METHOD testIsEqualToIgnoreCase : BOOL
VAR_INPUT
	(* for the test it's the parameter ``stringToCheck`` *)
	{attribute 'TcEncoding' := 'UTF-8'}
	stringToTest 	:Tc2_System.T_MaxString;
	(* for the test it's the parameter ``expected`` *)
	{attribute 'TcEncoding' := 'UTF-8'}
	expectedString	:Tc2_System.T_MaxString;
END_VAR
VAR 
	(* just the expectation if the assertion to test must be worng or true *)
	assertionIsWrong				:BOOL;
	(* contains the format string for the test message *)
	message							:Tc2_System.T_MaxString;
	(* contains ´´stringToTest´´ in upper case *)
	upperStringToTest				:Tc2_System.T_MaxString;
	(* contains ´´expectedString´´ in upper case *)
	upperExpectedString				:Tc2_System.T_MaxString;
	(* used for placeholder string if stringToTest can't be printed *)
	stringToTestAsString 			:Tc2_System.T_MaxString;
	(* used for placeholder string if expectedString can't be printed *)
	expectedStringAsString 			:Tc2_System.T_MaxString;
	(* contains stringToTest in normalized form *)
	normalizedStringToTest			:Tc2_System.T_MaxString;
	(* contains expectedString in normalized form *)
	normalizedExpectedString		:Tc2_System.T_MaxString;
	(* contains stringToTest in normalized form in upper case*)
	normalizedUpperStringToTest		:Tc2_System.T_MaxString;
	(* contains expectedString in normalized form in upper case*)
	normalizedUpperExpectedString	:Tc2_System.T_MaxString;
	(* holds characterCount of ``stringToTest`` *)
	stringToTestCharacterCount		:UDINT;
	(* holds characterCount of ``expectedString`` *)
	expectedCharacterCount			:UDINT;
	(* TwinCAT printf with the test message *)
	messageStringBuilder			:Tc2_Utilities.FB_FormatString;
	(* hold stringToCheck before assertion *)
	stringToTestBeforeAssertion		:Tc2_System.T_MaxString;
	(* hold expectedString before assertion *)
	expectedStringBeforeAssertion	:Tc2_System.T_MaxString;
END_VAR
THIS^.assertorContainer.resetAssertor();

stringToTestBeforeAssertion := stringToTest;
expectedStringBeforeAssertion := expectedString;
stringToTestAsString := stringToTest;
expectedStringAsString := expectedString;
upperStringToTest := stringToTest;
upperExpectedString := expectedString;

// both Strings to upper case
CNM_UnicodeUtilities.UpperCaseUtf8(ADR(upperStringToTest));
CNM_UnicodeUtilities.UpperCaseUtf8(ADR(upperExpectedString));

CNM_UnicodeUtilities.GetUtf8StringLength(
	ADR(upperStringToTest),
	characterCount => stringToTestCharacterCount
);
CNM_UnicodeUtilities.GetUtf8StringLength(
	ADR(upperExpectedString),
	characterCount => expectedCharacterCount
);
assertionIsWrong := ((
		stringToTestCharacterCount <> expectedCharacterCount
	) OR (
		CNM_UnicodeUtilities.FindInUtf8String(
			ADR(upperStringToTest),
			ADR(upperExpectedString)
		) <> 1
	)
);

message := SEL(
	assertionIsWrong,
	'stringToCheck is $'%s$' expected is $'%s$' assertion must be TRUE', 
	'stringToCheck is $'%s$' expected is $'%s$' assertion must be FALSE'
);

IF (
		Tc2_Standard.LEN(stringToTest) = TO_UINT(Tc2_System.MAX_STRING_LENGTH)
) THEN
	stringToTestAsString := 'String with Tc2_System.MAX_STRING_LENGTH characters';
END_IF
IF (
		Tc2_Standard.LEN(expectedString) = TO_UINT(Tc2_System.MAX_STRING_LENGTH)
) THEN
	expectedStringAsString := 'String with Tc2_System.MAX_STRING_LENGTH characters';
END_IF

messageStringBuilder(
	sFormat := message,
	arg1 := THIS^.AnyToArg(stringToTestAsString),
	arg2 := THIS^.AnyToArg(expectedStringAsString)
);


THIS^.assertorContainer.assertor.assert.strings.unicode.isEqualTo(
	stringToCheck := stringToTest,
	expected := expectedString,
	ignoreCases := TRUE,
	normalizeStrings := FALSE,
	message			:= ''
);

THIS^.AssertEquals_BOOL(
	Expected 	:= assertionIsWrong,
	Actual 		:= THIS^.assertorContainer.wasAssertionWrong,
	Message 	:= messageStringBuilder.sOut
);

THIS^.AssertEquals_STRING(
	Expected 	:= stringToTestBeforeAssertion,
	Actual 		:= stringToTest,
	Message 	:= 'the assertion changed $'stringToTest$''
);

THIS^.AssertEquals_STRING(
	Expected 	:= expectedStringBeforeAssertion,
	Actual 		:= expectedString,
	Message 	:= 'the assertion changed $'expectedString$''
);

THIS^.assertorContainer.resetAssertor();

CNM_UnicodeUtilities.NormalizeUtf8String(
	utf8StringBuffer := ADR(stringToTest),
	bufferSize := Tc2_System.MAX_STRING_LENGTH + 1,
	normalizedStringBuffer := ADR(normalizedStringToTest),
	normalForm := CNM_UnicodeUtilities.NormalizationForm.NFD
);
CNM_UnicodeUtilities.NormalizeUtf8String(
	utf8StringBuffer := ADR(expectedString),
	bufferSize := Tc2_System.MAX_STRING_LENGTH + 1,
	normalizedStringBuffer := ADR(normalizedExpectedString),
	normalForm := CNM_UnicodeUtilities.NormalizationForm.NFD
);

normalizedUpperStringToTest := normalizedStringToTest;
normalizedUpperExpectedString := normalizedExpectedString;
CNM_UnicodeUtilities.UpperCaseUtf8(ADR(normalizedUpperStringToTest));
CNM_UnicodeUtilities.UpperCaseUtf8(ADR(normalizedUpperExpectedString));

CNM_UnicodeUtilities.GetUtf8StringLength(
	ADR(normalizedUpperStringToTest),
	characterCount => stringToTestCharacterCount
);
CNM_UnicodeUtilities.GetUtf8StringLength(
	ADR(normalizedUpperExpectedString),
	characterCount => expectedCharacterCount
);
assertionIsWrong := ((
		stringToTestCharacterCount <> expectedCharacterCount
	) OR (
		CNM_UnicodeUtilities.FindInUtf8String(
			ADR(normalizedUpperStringToTest),
			ADR(normalizedUpperExpectedString)
		) <> 1
	)
);

THIS^.assertorContainer.assertor.assert.strings.unicode.isEqualTo(
	stringToCheck := stringToTest,
	expected := expectedString,
	ignoreCases := TRUE,
	normalizeStrings := TRUE,
	message			:= ''
);

THIS^.AssertEquals_BOOL(
	Expected 	:= assertionIsWrong,
	Actual 		:= THIS^.assertorContainer.wasAssertionWrong,
	Message 	:= messageStringBuilder.sOut
);

THIS^.AssertEquals_STRING(
	Expected 	:= stringToTestBeforeAssertion,
	Actual 		:= stringToTest,
	Message 	:= 'the assertion changed $'stringToTest$''
);

THIS^.AssertEquals_STRING(
	Expected 	:= expectedStringBeforeAssertion,
	Actual 		:= expectedString,
	Message 	:= 'the assertion changed $'expectedString$''
);
END_METHOD

(*
short summary
==================
This test method tests ``assert.string.unicode.isNotEmpty``
method of CNM_AssertionInterfaces library with various inputs

.. <legal notes>

legal notes
=================
| SPDX-FileCopyrightText: © 2022 ekvip automation GmbH <info@ekvip.de>
| SPDX-License-Identifier: Apache-2.0
| For details check: Apache-2.0_

.. _Apache-2.0: https://www.apache.org/licenses/LICENSE-2.0

.. </legal notes>

*)


METHOD testIsNotEmpty : BOOL
VAR_INPUT
	(* for the test it's the parameter ``stringToCheck`` *)
	{attribute 'TcEncoding' := 'UTF-8'}
	stringToTest :Tc2_System.T_MaxString;
END_VAR
VAR 
	(* just the expectation if the assertion to test must be worng or true *)
	assertionIsWrong				:BOOL;
	(* contains the format string for the test message *)
	message							:Tc2_System.T_MaxString;
	(* used for placeholder string if stringToTest can't be printed *)
	stringToTestAsString 			:Tc2_System.T_MaxString;
	(* holds characterCount of ``stringToTest`` *)
	stringToTestCharacterCount		:UDINT;
	(* TwinCAT printf with the test message *)
	messageStringBuilder			:Tc2_Utilities.FB_FormatString;
	(* hold stringToCheck before assertion *)
	stringToTestBeforeAssertion		:Tc2_System.T_MaxString;
END_VAR
THIS^.assertorContainer.resetAssertor();

stringToTestBeforeAssertion := stringToTest;
stringToTestAsString := stringToTest;

CNM_UnicodeUtilities.GetUtf8StringLength(
	ADR(stringToTest),
	characterCount => stringToTestCharacterCount
);
assertionIsWrong :=  stringToTestCharacterCount = 0;

message := SEL(
	assertionIsWrong,
	'stringToCheck is $'%s$' assertion must be TRUE', 
	'stringToCheck is $'%s$' assertion must be FALSE'
);

IF (
		Tc2_Standard.LEN(stringToTest) = TO_UINT(Tc2_System.MAX_STRING_LENGTH)
) THEN
	stringToTestAsString := 'String with Tc2_System.MAX_STRING_LENGTH characters';
END_IF

messageStringBuilder(
	sFormat := message,
	arg1 := THIS^.AnyToArg(stringToTestAsString),
);


THIS^.assertorContainer.assertor.assert.strings.unicode.isNotEmpty(
	stringToCheck := stringToTest,
	message			:= ''
);

THIS^.AssertEquals_BOOL(
	Expected 	:= assertionIsWrong,
	Actual 		:= THIS^.assertorContainer.wasAssertionWrong,
	Message 	:= messageStringBuilder.sOut
);

THIS^.AssertEquals_STRING(
	Expected 	:= stringToTestBeforeAssertion,
	Actual 		:= stringToTest,
	Message 	:= 'the assertion changed $'stringToTest$''
);
END_METHOD

(*
short summary
==================
This test method tests ``assert.string.unicode.isNotEqualTo``
method of CNM_AssertionInterfaces library with various inputs

.. <legal notes>

legal notes
=================
| SPDX-FileCopyrightText: © 2022 ekvip automation GmbH <info@ekvip.de>
| SPDX-License-Identifier: Apache-2.0
| For details check: Apache-2.0_

.. _Apache-2.0: https://www.apache.org/licenses/LICENSE-2.0

.. </legal notes>

*)


METHOD testIsNotEqualTo : BOOL
VAR_INPUT
	(* for the test it's the parameter ``stringToCheck`` *)
	{attribute 'TcEncoding' := 'UTF-8'}
	stringToTest 	:Tc2_System.T_MaxString;
	(* for the test it's the parameter ``unexpected`` *)
	{attribute 'TcEncoding' := 'UTF-8'}
	expectedString :Tc2_System.T_MaxString;
END_VAR
VAR 
	(* just the expectation if the assertion to test must be worng or true *)
	assertionIsWrong				:BOOL;
	(* contains the format string for the test message *)
	message							:Tc2_System.T_MaxString;
	(* used for placeholder string if stringToTest can't be printed *)
	stringToTestAsString 			:Tc2_System.T_MaxString;
	(* used for placeholder string if expectedString can't be printed *)
	expectedStringAsString 			:Tc2_System.T_MaxString;
	(* contains stringToTest in normalized form *)
	normalizedStringToTest			:Tc2_System.T_MaxString;
	(* contains expectedString in normalized form *)
	normalizedExpectedString		:Tc2_System.T_MaxString;
	(* holds characterCount of ``stringToTest`` *)
	stringToTestCharacterCount		:UDINT;
	(* holds characterCount of ``expectedString`` *)
	expectedCharacterCount			:UDINT;
	(* TwinCAT printf with the test message *)
	messageStringBuilder			:Tc2_Utilities.FB_FormatString;
	(* hold stringToCheck before assertion *)
	stringToTestBeforeAssertion		:Tc2_System.T_MaxString;
	(* hold expectedString before assertion *)
	expectedStringBeforeAssertion	:Tc2_System.T_MaxString;
	expected: INT;
END_VAR
THIS^.assertorContainer.resetAssertor();

stringToTestBeforeAssertion := stringToTest;
expectedStringBeforeAssertion := expectedString;
stringToTestAsString := stringToTest;
expectedStringAsString := expectedString;

CNM_UnicodeUtilities.GetUtf8StringLength(
	ADR(stringToTest),
	characterCount => stringToTestCharacterCount
);
CNM_UnicodeUtilities.GetUtf8StringLength(
	ADR(expectedString),
	characterCount => expectedCharacterCount
);
assertionIsWrong := ((
		stringToTestCharacterCount = expectedCharacterCount
	) AND_THEN (
		CNM_UnicodeUtilities.FindInUtf8String(
			ADR(stringToTest),
			ADR(expectedString)
		) = 1
	)
);

message := SEL(
	assertionIsWrong,
	'stringToCheck is $'%s$' unexpected is $'%s$' assertion must be TRUE', 
	'stringToCheck is $'%s$' unexpected is $'%s$' assertion must be FALSE'
);

IF (
		Tc2_Standard.LEN(stringToTest) = TO_UINT(Tc2_System.MAX_STRING_LENGTH)
) THEN
	stringToTestAsString := 'String with Tc2_System.MAX_STRING_LENGTH characters';
END_IF
IF (
		Tc2_Standard.LEN(expectedString) = TO_UINT(Tc2_System.MAX_STRING_LENGTH)
) THEN
	expectedStringAsString := 'String with Tc2_System.MAX_STRING_LENGTH characters';
END_IF


messageStringBuilder(
	sFormat := message,
	arg1 := THIS^.AnyToArg(stringToTestAsString),
	arg2 := THIS^.AnyToArg(expectedStringAsString)
);


THIS^.assertorContainer.assertor.assert.strings.unicode.isNotEqualTo(
	stringToCheck := stringToTest,
	unexpected := expectedString,
	ignoreCases := FALSE,
	normalizeStrings := FALSE,
	message			:= ''
);

THIS^.AssertEquals_BOOL(
	Expected 	:= assertionIsWrong,
	Actual 		:= THIS^.assertorContainer.wasAssertionWrong,
	Message 	:= messageStringBuilder.sOut
);

THIS^.AssertEquals_STRING(
	Expected 	:= stringToTestBeforeAssertion,
	Actual 		:= stringToTest,
	Message 	:= 'the assertion changed $'stringToTest$''
);

THIS^.AssertEquals_STRING(
	Expected 	:= expectedStringBeforeAssertion,
	Actual 		:= expectedString,
	Message 	:= 'the assertion changed $'expectedString$''
);

THIS^.assertorContainer.resetAssertor();

CNM_UnicodeUtilities.NormalizeUtf8String(
	utf8StringBuffer := ADR(stringToTest),
	bufferSize := Tc2_System.MAX_STRING_LENGTH + 1,
	normalizedStringBuffer := ADR(normalizedStringToTest),
	normalForm := CNM_UnicodeUtilities.NormalizationForm.NFD
);
CNM_UnicodeUtilities.NormalizeUtf8String(
	utf8StringBuffer := ADR(expectedString),
	bufferSize := Tc2_System.MAX_STRING_LENGTH + 1,
	normalizedStringBuffer := ADR(normalizedExpectedString),
	normalForm := CNM_UnicodeUtilities.NormalizationForm.NFD
);

CNM_UnicodeUtilities.GetUtf8StringLength(
	ADR(normalizedStringToTest),
	characterCount => stringToTestCharacterCount
);
CNM_UnicodeUtilities.GetUtf8StringLength(
	ADR(normalizedExpectedString),
	characterCount => expectedCharacterCount
);
assertionIsWrong := ((
		stringToTestCharacterCount = expectedCharacterCount
	) AND (
		CNM_UnicodeUtilities.FindInUtf8String(
			ADR(normalizedStringToTest),
			ADR(normalizedExpectedString)
		) = 1
	)
);

THIS^.assertorContainer.assertor.assert.strings.unicode.isNotEqualTo(
	stringToCheck := stringToTest,
	unexpected := expectedString,
	ignoreCases := FALSE,
	normalizeStrings := TRUE,
	message			:= ''
);

THIS^.AssertEquals_BOOL(
	Expected 	:= assertionIsWrong,
	Actual 		:= THIS^.assertorContainer.wasAssertionWrong,
	Message 	:= messageStringBuilder.sOut
);

THIS^.AssertEquals_STRING(
	Expected 	:= stringToTestBeforeAssertion,
	Actual 		:= stringToTest,
	Message 	:= 'the assertion changed $'stringToTest$''
);

THIS^.AssertEquals_STRING(
	Expected 	:= expectedStringBeforeAssertion,
	Actual 		:= expectedString,
	Message 	:= 'the assertion changed $'expectedString$''
);
END_METHOD

(*
short summary
==================
This test method tests ``assert.string.unicode.isNotEqualTo``
method of CNM_AssertionInterfaces library with various inputs

.. <legal notes>

legal notes
=================
| SPDX-FileCopyrightText: © 2022 ekvip automation GmbH <info@ekvip.de>
| SPDX-License-Identifier: Apache-2.0
| For details check: Apache-2.0_

.. _Apache-2.0: https://www.apache.org/licenses/LICENSE-2.0

.. </legal notes>

*)


METHOD testIsNotEqualToIgnoreCase : BOOL
VAR_INPUT
	(* for the test it's the parameter ``stringToCheck`` *)
	{attribute 'TcEncoding' := 'UTF-8'}
	stringToTest 	:Tc2_System.T_MaxString;
	(* for the test it's the parameter ``unexpected`` *)
	{attribute 'TcEncoding' := 'UTF-8'}
	expectedString :Tc2_System.T_MaxString;
END_VAR
VAR 
	(* just the expectation if the assertion to test must be worng or true *)
	assertionIsWrong				:BOOL;
	(* contains the format string for the test message *)
	message							:Tc2_System.T_MaxString;
	(* contains ´´stringToTest´´ in upper case *)
	upperStringToTest				:Tc2_System.T_MaxString;
	(* contains ´´expectedString´´ in upper case *)
	upperExpectedString				:Tc2_System.T_MaxString;
	(* used for placeholder string if stringToTest can't be printed *)
	stringToTestAsString 			:Tc2_System.T_MaxString;
	(* used for placeholder string if expectedString can't be printed *)
	expectedStringAsString 			:Tc2_System.T_MaxString;
	(* contains stringToTest in normalized form *)
	normalizedStringToTest			:Tc2_System.T_MaxString;
	(* contains expectedString in normalized form *)
	normalizedExpectedString		:Tc2_System.T_MaxString;
	(* contains stringToTest in normalized form in upper case*)
	normalizedUpperStringToTest		:Tc2_System.T_MaxString;
	(* contains expectedString in normalized form in upper case*)
	normalizedUpperExpectedString	:Tc2_System.T_MaxString;
	(* holds characterCount of ``stringToTest`` *)
	stringToTestCharacterCount		:UDINT;
	(* holds characterCount of ``expectedString`` *)
	expectedCharacterCount			:UDINT;
	(* TwinCAT printf with the test message *)
	messageStringBuilder			:Tc2_Utilities.FB_FormatString;
	(* hold stringToCheck before assertion *)
	stringToTestBeforeAssertion		:Tc2_System.T_MaxString;
	(* hold expectedString before assertion *)
	expectedStringBeforeAssertion	:Tc2_System.T_MaxString;
END_VAR
THIS^.assertorContainer.resetAssertor();

stringToTestBeforeAssertion := stringToTest;
expectedStringBeforeAssertion := expectedString;
stringToTestAsString := stringToTest;
expectedStringAsString := expectedString;
upperStringToTest := stringToTest;
upperExpectedString := expectedString;

// both Strings to upper case
CNM_UnicodeUtilities.UpperCaseUtf8(ADR(upperStringToTest));
CNM_UnicodeUtilities.UpperCaseUtf8(ADR(upperExpectedString));

CNM_UnicodeUtilities.GetUtf8StringLength(
	ADR(upperStringToTest),
	characterCount => stringToTestCharacterCount
);
CNM_UnicodeUtilities.GetUtf8StringLength(
	ADR(upperExpectedString),
	characterCount => expectedCharacterCount
);
assertionIsWrong := ((
		stringToTestCharacterCount = expectedCharacterCount
	) AND (
		CNM_UnicodeUtilities.FindInUtf8String(
			ADR(upperStringToTest),
			ADR(upperExpectedString)
		) = 1
	)
);

message := SEL(
	assertionIsWrong,
	'stringToCheck is $'%s$' unexpected is $'%s$' assertion must be TRUE', 
	'stringToCheck is $'%s$' unexpected is $'%s$' assertion must be FALSE'
);

IF (
		Tc2_Standard.LEN(stringToTest) = TO_UINT(Tc2_System.MAX_STRING_LENGTH)
) THEN
	stringToTestAsString := 'String with Tc2_System.MAX_STRING_LENGTH characters';
END_IF
IF (
		Tc2_Standard.LEN(expectedString) = TO_UINT(Tc2_System.MAX_STRING_LENGTH)
) THEN
	expectedStringAsString := 'String with Tc2_System.MAX_STRING_LENGTH characters';
END_IF

messageStringBuilder(
	sFormat := message,
	arg1 := THIS^.AnyToArg(stringToTestAsString),
	arg2 := THIS^.AnyToArg(expectedStringAsString)
);


THIS^.assertorContainer.assertor.assert.strings.unicode.isNotEqualTo(
	stringToCheck := stringToTest,
	unexpected := expectedString,
	ignoreCases := TRUE,
	normalizeStrings := FALSE,
	message			:= ''
);

THIS^.AssertEquals_BOOL(
	Expected 	:= assertionIsWrong,
	Actual 		:= THIS^.assertorContainer.wasAssertionWrong,
	Message 	:= messageStringBuilder.sOut
);

THIS^.AssertEquals_STRING(
	Expected 	:= stringToTestBeforeAssertion,
	Actual 		:= stringToTest,
	Message 	:= 'the assertion changed $'stringToTest$''
);

THIS^.AssertEquals_STRING(
	Expected 	:= expectedStringBeforeAssertion,
	Actual 		:= expectedString,
	Message 	:= 'the assertion changed $'expectedString$''
);

THIS^.assertorContainer.resetAssertor();

CNM_UnicodeUtilities.NormalizeUtf8String(
	utf8StringBuffer := ADR(stringToTest),
	bufferSize := Tc2_System.MAX_STRING_LENGTH + 1,
	normalizedStringBuffer := ADR(normalizedStringToTest),
	normalForm := CNM_UnicodeUtilities.NormalizationForm.NFD
);
CNM_UnicodeUtilities.NormalizeUtf8String(
	utf8StringBuffer := ADR(expectedString),
	bufferSize := Tc2_System.MAX_STRING_LENGTH + 1,
	normalizedStringBuffer := ADR(normalizedExpectedString),
	normalForm := CNM_UnicodeUtilities.NormalizationForm.NFD
);

normalizedUpperStringToTest := normalizedStringToTest;
normalizedUpperExpectedString := normalizedExpectedString;
CNM_UnicodeUtilities.UpperCaseUtf8(ADR(normalizedUpperStringToTest));
CNM_UnicodeUtilities.UpperCaseUtf8(ADR(normalizedUpperExpectedString));

CNM_UnicodeUtilities.GetUtf8StringLength(
	ADR(normalizedUpperStringToTest),
	characterCount => stringToTestCharacterCount
);
CNM_UnicodeUtilities.GetUtf8StringLength(
	ADR(normalizedUpperExpectedString),
	characterCount => expectedCharacterCount
);
assertionIsWrong := ((
		stringToTestCharacterCount = expectedCharacterCount
	) AND (
		CNM_UnicodeUtilities.FindInUtf8String(
			ADR(normalizedUpperStringToTest),
			ADR(normalizedUpperExpectedString)
		) = 1
	)
);

THIS^.assertorContainer.assertor.assert.strings.unicode.isNotEqualTo(
	stringToCheck := stringToTest,
	unexpected := expectedString,
	ignoreCases := TRUE,
	normalizeStrings := TRUE,
	message			:= ''
);

THIS^.AssertEquals_BOOL(
	Expected 	:= assertionIsWrong,
	Actual 		:= THIS^.assertorContainer.wasAssertionWrong,
	Message 	:= messageStringBuilder.sOut
);

THIS^.AssertEquals_STRING(
	Expected 	:= stringToTestBeforeAssertion,
	Actual 		:= stringToTest,
	Message 	:= 'the assertion changed $'stringToTest$''
);

THIS^.AssertEquals_STRING(
	Expected 	:= expectedStringBeforeAssertion,
	Actual 		:= expectedString,
	Message 	:= 'the assertion changed $'expectedString$''
);
END_METHOD

(*
short summary
==================
This test method tests ``assert.string.unicode.lengthIsBetween``
method of CNM_AssertionInterfaces library with various inputs

.. <legal notes>

legal notes
=================
| SPDX-FileCopyrightText: © 2022 ekvip automation GmbH <info@ekvip.de>
| SPDX-License-Identifier: Apache-2.0
| For details check: Apache-2.0_

.. _Apache-2.0: https://www.apache.org/licenses/LICENSE-2.0

.. </legal notes>

*)


METHOD testLengthIsBetween : BOOL
VAR_INPUT
	(* for the test it's the parameter ``stringToCheck`` *)
	{attribute 'TcEncoding' := 'UTF-8'}
	stringToTest 			:Tc2_System.T_MaxString;
	(* for the test it's the parameter ``maxLength`` *)
	maxLength 				:UDINT;
	(* for the test it's the parameter ``minLength`` *)
	minLength 				:UDINT;
	(* UnicodeStringLengthUnit the input is tested for *)
	stringLengthUnit		:CNM_AssertionInterfaces.UnicodeStringLengthUnit;
	(* contains ``stringToTest`` in only ascii charachters for test output *)
	stringToTestPrintable 	:Tc2_System.T_MaxString := '';
END_VAR
VAR 
	(* just the expectation if the assertion to test must be worng or true *)
	assertionIsWrong				:BOOL;
	(* contains the format string for the test message *)
	message							:Tc2_System.T_MaxString;
	(* used for placeholder string if stringToTest can't be printed *)
	stringToTestAsString 			:Tc2_System.T_MaxString;
	(* holds string with current ´´stringLengthUnit´´ for the test message*)
	currentStringLengthUnit 		:Tc2_System.T_MaxString;
	(* TwinCAT printf with the test message *)
	messageStringBuilder			:Tc2_Utilities.FB_FormatString;
	(* length of current string to check in bytes *)
	stringToTestByteCount			:UDINT;
	(* length of current string to check in characters *)
	stringToTestCodePointCount		:UDINT;
	(* length of ´´stringToCheck´´ *)
	normalizedLength 				:UDINT;
	(* holds the normalized ´´stringToCheck´´ *)
	{attribute 'TcEncoding' := 'UTF-8'}
	normalizedStringToTest 			:Tc2_System.T_MaxString;
	(* width of ´´stringToCheck´´ *)
	stringToTestWidth 				:DINT;
	(* visible characters of ´´stringToCheck´´ *)
	stringToTestVisibleCharacters	:UDINT := 0;
	(* hold stringToCheck before assertion *)
	stringToTestBeforeAssertion		:Tc2_System.T_MaxString;
END_VAR
THIS^.assertorContainer.resetAssertor();

stringToTestBeforeAssertion := stringToTest;
stringToTestAsString := stringToTest;

CNM_UnicodeUtilities.GetUtf8StringLength(ADR(stringToTest), byteCount => stringToTestByteCount, characterCount => stringToTestCodePointCount,);
CNM_UnicodeUtilities.GetUtf8StringWidth(ADR(stringToTest), visibleCharacters => stringToTestVisibleCharacters, width => stringToTestWidth);

IF (
		Tc2_Standard.LEN(stringToTest) = TO_UINT(Tc2_System.MAX_STRING_LENGTH)
) THEN
	stringToTestAsString := 'String with Tc2_System.MAX_STRING_LENGTH characters';
END_IF
IF (
		LEN(stringToTestPrintable) <> 0
) THEN
	stringToTestAsString := stringToTestPrintable;
END_IF

CASE stringLengthUnit OF
	
CNM_AssertionInterfaces.UnicodeStringLengthUnit.BYTES:
	currentStringLengthUnit := 'BYTES';
	
	assertionIsWrong := ((stringToTestByteCount < minLength) OR ( stringToTestByteCount > maxLength ));
	
	message := SEL(
		assertionIsWrong,
		'stringToCheck is $'%s$' with maxLength %u and minLength %u assertion must be TRUE  (%S)', 
		'stringToCheck is $'%s$' with maxLength %u and minLength %u assertion must be FALSE  (%S)'
	);
	
	messageStringBuilder(
		sFormat := message,
		arg1 := THIS^.AnyToArg(stringToTestAsString),
		arg2 := THIS^.AnyToArg(maxLength),
		arg3 := THIS^.AnyToArg(minLength),
		arg4 := THIS^.AnyToArg(currentStringLengthUnit)
	);
	
	THIS^.assertorContainer.assertor.assert.strings.unicode.lengthIsBetween(
		stringToCheck := stringToTest,
		maxLength := maxLength,
		minLength := minLength,
		stringLengthUnit := CNM_AssertionInterfaces.UnicodeStringLengthUnit.BYTES,
		message			:= ''
	);
	
	THIS^.AssertEquals_BOOL(
		Expected 	:= assertionIsWrong,
		Actual 		:= THIS^.assertorContainer.wasAssertionWrong,
		Message 	:= messageStringBuilder.sOut
	);
	
	THIS^.AssertEquals_STRING(
		Expected 	:= stringToTestBeforeAssertion,
		Actual 		:= stringToTest,
		Message 	:= 'the assertion changed $'stringToTest$''
	);
	
CNM_AssertionInterfaces.UnicodeStringLengthUnit.CHARACTERS:	
	currentStringLengthUnit := 'CHARACTERS';
	THIS^.assertorContainer.resetAssertor();
	
	assertionIsWrong := ((
			stringToTestCodePointCount < minLength
		) OR (
			stringToTestCodePointCount > maxLength
		)
	);
	
	message := SEL(
		assertionIsWrong,
		'stringToCheck is $'%s$' with maxLength %u and minLength %u assertion must be TRUE  (%S)', 
		'stringToCheck is $'%s$' with maxLength %u and minLength %u assertion must be FALSE  (%S)'
	);
	
	   messageStringBuilder(
		sFormat := message,
		arg1 := THIS^.AnyToArg(stringToTestAsString),
		arg2 := THIS^.AnyToArg(maxLength),
		arg3 := THIS^.AnyToArg(minLength),
		arg4 := THIS^.AnyToArg(currentStringLengthUnit)
	);
	
	THIS^.assertorContainer.assertor.assert.strings.unicode.lengthIsBetween(
		stringToCheck := stringToTest,
		maxLength := maxLength,
		minLength := minLength,
		stringLengthUnit := CNM_AssertionInterfaces.UnicodeStringLengthUnit.CHARACTERS,
		message			:= ''
	);
	
	THIS^.AssertEquals_BOOL(
		Expected 	:= assertionIsWrong,
		Actual 		:= THIS^.assertorContainer.wasAssertionWrong,
		Message 	:= messageStringBuilder.sOut
	);
	
	THIS^.AssertEquals_STRING(
		Expected 	:= stringToTestBeforeAssertion,
		Actual 		:= stringToTest,
		Message 	:= 'the assertion changed $'stringToTest$''
	);
	
CNM_AssertionInterfaces.UnicodeStringLengthUnit.CHARACTERS_NFD:	
	currentStringLengthUnit := 'NFD';
	THIS^.assertorContainer.resetAssertor();
	
	CNM_UnicodeUtilities.NormalizeUtf8String(
		utf8StringBuffer := ADR(stringToTest),
		normalForm := CNM_UnicodeUtilities.NormalizationForm.NFD,
		normalizedStringBuffer := ADR(normalizedStringToTest),
		bufferSize := Tc2_System.MAX_STRING_LENGTH + 1,
		normalizedStringLength => normalizedLength
	);
	CNM_UnicodeUtilities.GetUtf8StringLength(
		stringAddress := ADR(normalizedStringToTest),
		characterCount => stringToTestCodePointCount
	);
		
	assertionIsWrong := ((
			stringToTestCodePointCount < minLength
		) OR (
			stringToTestCodePointCount > maxLength
		)
	);
	
	message := SEL(
		assertionIsWrong,
		'stringToCheck is $'%s$' with maxLength %u and minLength %u assertion must be TRUE  (%S)', 
		'stringToCheck is $'%s$' with maxLength %u and minLength %u assertion must be FALSE  (%S)'
	);
	
	messageStringBuilder(
		sFormat := message,
		arg1 := THIS^.AnyToArg(stringToTestAsString),
		arg2 := THIS^.AnyToArg(maxLength),
		arg3 := THIS^.AnyToArg(minLength),
		arg4 := THIS^.AnyToArg(currentStringLengthUnit)
	);
	
	THIS^.assertorContainer.assertor.assert.strings.unicode.lengthIsBetween(
		stringToCheck := stringToTest,
		maxLength := maxLength,
		minLength := minLength,
		stringLengthUnit := CNM_AssertionInterfaces.UnicodeStringLengthUnit.CHARACTERS_NFD,
		message			:= ''
	);
	
	THIS^.AssertEquals_BOOL(
		Expected 	:= assertionIsWrong,
		Actual 		:= THIS^.assertorContainer.wasAssertionWrong,
		Message 	:= messageStringBuilder.sOut
	);
	
	THIS^.AssertEquals_STRING(
		Expected 	:= stringToTestBeforeAssertion,
		Actual 		:= stringToTest,
		Message 	:= 'the assertion changed $'stringToTest$''
	);
	
CNM_AssertionInterfaces.UnicodeStringLengthUnit.CHARACTERS_NFC:	
	currentStringLengthUnit := 'NFC';
	THIS^.assertorContainer.resetAssertor();
	
	CNM_UnicodeUtilities.NormalizeUtf8String(
		utf8StringBuffer := ADR(stringToTest),
		normalForm := CNM_UnicodeUtilities.NormalizationForm.NFC,
		normalizedStringBuffer := ADR(normalizedStringToTest),
		bufferSize := Tc2_System.MAX_STRING_LENGTH + 1,
		normalizedStringLength => normalizedLength
	);
	CNM_UnicodeUtilities.GetUtf8StringLength(
		stringAddress := ADR(normalizedStringToTest),
		characterCount => stringToTestCodePointCount
	);
		
	assertionIsWrong := ((
			stringToTestCodePointCount < minLength
		) OR (
			stringToTestCodePointCount > maxLength
		)
	);
	
	message := SEL(
		assertionIsWrong,
		'stringToCheck is $'%s$' with maxLength %u and minLength %u assertion must be TRUE  (%S)', 
		'stringToCheck is $'%s$' with maxLength %u and minLength %u assertion must be FALSE  (%S)'
	);
	
	messageStringBuilder(
		sFormat := message,
		arg1 := THIS^.AnyToArg(stringToTestAsString),
		arg2 := THIS^.AnyToArg(maxLength),
		arg3 := THIS^.AnyToArg(minLength),
		arg4 := THIS^.AnyToArg(currentStringLengthUnit)
	);
	
	THIS^.assertorContainer.assertor.assert.strings.unicode.lengthIsBetween(
		stringToCheck := stringToTest,
		maxLength := maxLength,
		minLength := minLength,
		stringLengthUnit := CNM_AssertionInterfaces.UnicodeStringLengthUnit.CHARACTERS_NFC,
		message			:= ''
	);
	
	THIS^.AssertEquals_BOOL(
		Expected 	:= assertionIsWrong,
		Actual 		:= THIS^.assertorContainer.wasAssertionWrong,
		Message 	:= messageStringBuilder.sOut
	);
	
	THIS^.AssertEquals_STRING(
		Expected 	:= stringToTestBeforeAssertion,
		Actual 		:= stringToTest,
		Message 	:= 'the assertion changed $'stringToTest$''
	);
	
CNM_AssertionInterfaces.UnicodeStringLengthUnit.VISIBLE_CHARACTERS:	
	currentStringLengthUnit := 'VISIBLE_CHARACTERS';
	THIS^.assertorContainer.resetAssertor();
	
	assertionIsWrong := ((
			stringToTestVisibleCharacters < minLength
		) OR (
			stringToTestVisibleCharacters > maxLength
		)
	);
	
	message := SEL(
		assertionIsWrong,
		'stringToCheck is $'%s$' with maxLength %u and minLength %u assertion must be TRUE  (%S)', 
		'stringToCheck is $'%s$' with maxLength %u and minLength %u assertion must be FALSE  (%S)'
	);
	
	messageStringBuilder(
		sFormat := message,
		arg1 := THIS^.AnyToArg(stringToTestAsString),
		arg2 := THIS^.AnyToArg(maxLength),
		arg3 := THIS^.AnyToArg(minLength),
		arg4 := THIS^.AnyToArg(currentStringLengthUnit)
	);
	
	THIS^.assertorContainer.assertor.assert.strings.unicode.lengthIsBetween(
		stringToCheck := stringToTest,
		maxLength := maxLength,
		minLength := minLength,
		stringLengthUnit := CNM_AssertionInterfaces.UnicodeStringLengthUnit.VISIBLE_CHARACTERS,
		message			:= ''
	);
	
	THIS^.AssertEquals_BOOL(
		Expected 	:= assertionIsWrong,
		Actual 		:= THIS^.assertorContainer.wasAssertionWrong,
		Message 	:= messageStringBuilder.sOut
	);
	
	THIS^.AssertEquals_STRING(
		Expected 	:= stringToTestBeforeAssertion,
		Actual 		:= stringToTest,
		Message 	:= 'the assertion changed $'stringToTest$''
	);
	
CNM_AssertionInterfaces.UnicodeStringLengthUnit.WIDTH:	
	currentStringLengthUnit := 'WIDTH';
	THIS^.assertorContainer.resetAssertor();
	
	assertionIsWrong := ((
			TO_UDINT(stringToTestWidth) < minLength
		) OR (
			TO_UDINT(stringToTestWidth) > maxLength
		)
	);
	
	message := SEL(
		assertionIsWrong,
		'stringToCheck is $'%s$' with maxLength %u and minLength %u assertion must be TRUE  (%S)', 
		'stringToCheck is $'%s$' with maxLength %u and minLength %u assertion must be FALSE  (%S)'
	);
	
	messageStringBuilder(
		sFormat := message,
		arg1 := THIS^.AnyToArg(stringToTestAsString),
		arg2 := THIS^.AnyToArg(maxLength),
		arg3 := THIS^.AnyToArg(minLength),
		arg4 := THIS^.AnyToArg(currentStringLengthUnit)
	);
	
	THIS^.assertorContainer.assertor.assert.strings.unicode.lengthIsBetween(
		stringToCheck := stringToTest,
		maxLength := maxLength,
		minLength := minLength,
		stringLengthUnit := CNM_AssertionInterfaces.UnicodeStringLengthUnit.WIDTH,
		message			:= ''
	);
	
	THIS^.AssertEquals_BOOL(
		Expected 	:= assertionIsWrong,
		Actual 		:= THIS^.assertorContainer.wasAssertionWrong,
		Message 	:= messageStringBuilder.sOut
	);

	THIS^.AssertEquals_STRING(
		Expected 	:= stringToTestBeforeAssertion,
		Actual 		:= stringToTest,
		Message 	:= 'the assertion changed $'stringToTest$''
	);

END_CASE
END_METHOD

(*
short summary
==================
This test method tests ``assert.string.unicode.lengthIsExact``
method of CNM_AssertionInterfaces library with various inputs

.. <legal notes>

legal notes
=================
| SPDX-FileCopyrightText: © 2022 ekvip automation GmbH <info@ekvip.de>
| SPDX-License-Identifier: Apache-2.0
| For details check: Apache-2.0_

.. _Apache-2.0: https://www.apache.org/licenses/LICENSE-2.0

.. </legal notes>

*)


METHOD testLengthIsExact : BOOL
VAR_INPUT
	(* for the test it's the parameter ``stringToCheck`` *)
	{attribute 'TcEncoding' := 'UTF-8'}
	stringToTest 			:Tc2_System.T_MaxString;
	(* for the test it's the parameter ``expectedLength`` *)
	expectedLength			:UDINT;
	(* UnicodeStringLengthUnit the input is tested for *)
	stringLengthUnit		:CNM_AssertionInterfaces.UnicodeStringLengthUnit;
	(* contains ``stringToTest`` in only ascii charachters for test output *)
	stringToTestPrintable	:Tc2_System.T_MaxString := '';
END_VAR
VAR 
	(* just the expectation if the assertion to test must be worng or true *)
	assertionIsWrong				:BOOL;
	(* contains the format string for the test message *)
	message							:Tc2_System.T_MaxString;
	(* used for placeholder string if stringToTest can't be printed *)
	stringToTestAsString 			:Tc2_System.T_MaxString;
	(* holds string with current ´´stringLengthUnit´´ for the test message*)
	currentStringLengthUnit 		:Tc2_System.T_MaxString;
	(* TwinCAT printf with the test message *)
	messageStringBuilder			:Tc2_Utilities.FB_FormatString;
	(* length of current string to check in bytes *)
	stringToTestByteCount			:UDINT;
	(* length of current string to check in characters *)
	stringToTestCodePointCount		:UDINT;
	(* length of ´´stringToCheck´´ *)
	normalizedLength 				:UDINT;
	(* holds the normalized ´´stringToCheck´´ *)
	{attribute 'TcEncoding' := 'UTF-8'}
	normalizedStringToTest 			:Tc2_System.T_MaxString;
	(* width of ´´stringToCheck´´ *)
	stringToTestWidth 				:DINT;
	(* visible characters of ´´stringToCheck´´ *)
	stringToTestVisibleCharacters	:UDINT := 0;
	(* hold stringToCheck before assertion *)
	stringToTestBeforeAssertion		:Tc2_System.T_MaxString;
END_VAR
THIS^.assertorContainer.resetAssertor();

stringToTestBeforeAssertion := stringToTest;
stringToTestAsString := stringToTest;

CNM_UnicodeUtilities.GetUtf8StringLength(ADR(stringToTest), byteCount => stringToTestByteCount, characterCount => stringToTestCodePointCount,);
CNM_UnicodeUtilities.GetUtf8StringWidth(ADR(stringToTest), visibleCharacters => stringToTestVisibleCharacters, width => stringToTestWidth);

IF (
		Tc2_Standard.LEN(stringToTest) = TO_UINT(Tc2_System.MAX_STRING_LENGTH)
) THEN
	stringToTestAsString := 'String with Tc2_System.MAX_STRING_LENGTH characters';
END_IF
IF (
		LEN(stringToTestPrintable) <> 0
) THEN
	stringToTestAsString := stringToTestPrintable;
END_IF

CASE stringLengthUnit OF

CNM_AssertionInterfaces.UnicodeStringLengthUnit.BYTES:
	currentStringLengthUnit := 'BYTES';
	
	assertionIsWrong := stringToTestByteCount <> expectedLength;
	
	message := SEL(
		assertionIsWrong,
		'stringToCheck is $'%s$' with expectedLength %u assertion must be TRUE  (%S)', 
		'stringToCheck is $'%s$' with expectedLength %u assertion must be FALSE  (%S)'
	);
	
	messageStringBuilder(
		sFormat := message,
		arg1 := THIS^.AnyToArg(stringToTestAsString),
		arg2 := THIS^.AnyToArg(expectedLength),
		arg3 := THIS^.AnyToArg(currentStringLengthUnit)
	);
	
	THIS^.assertorContainer.assertor.assert.strings.unicode.lengthIsExact(
		stringToCheck := stringToTest,
		expectedLength := expectedLength,
		stringLengthUnit := CNM_AssertionInterfaces.UnicodeStringLengthUnit.BYTES,
		message			:= ''
	);
	
	THIS^.AssertEquals_BOOL(
		Expected 	:= assertionIsWrong,
		Actual 		:= THIS^.assertorContainer.wasAssertionWrong,
		Message 	:= messageStringBuilder.sOut
	);
	
	THIS^.AssertEquals_STRING(
		Expected 	:= stringToTestBeforeAssertion,
		Actual 		:= stringToTest,
		Message 	:= 'the assertion changed $'stringToTest$''
	);
	
CNM_AssertionInterfaces.UnicodeStringLengthUnit.CHARACTERS:	
	currentStringLengthUnit := 'CHARACTERS';
	
	assertionIsWrong := stringToTestCodePointCount <> expectedLength;
	
	message := SEL(
		assertionIsWrong,
		'stringToCheck is $'%s$' with expectedLength %u assertion must be TRUE  (%S)', 
		'stringToCheck is $'%s$' with expectedLength %u assertion must be FALSE  (%S)'
	);
	
	messageStringBuilder(
		sFormat := message,
		arg1 := THIS^.AnyToArg(stringToTestAsString),
		arg2 := THIS^.AnyToArg(expectedLength),
		arg3 := THIS^.AnyToArg(currentStringLengthUnit)
	);
	
	THIS^.assertorContainer.assertor.assert.strings.unicode.lengthIsExact(
		stringToCheck := stringToTest,
		expectedLength := expectedLength,
		stringLengthUnit := CNM_AssertionInterfaces.UnicodeStringLengthUnit.CHARACTERS,
		message			:= ''
	);
	
	THIS^.AssertEquals_BOOL(
		Expected 	:= assertionIsWrong,
		Actual 		:= THIS^.assertorContainer.wasAssertionWrong,
		Message 	:= messageStringBuilder.sOut
	);
	
	THIS^.AssertEquals_STRING(
		Expected 	:= stringToTestBeforeAssertion,
		Actual 		:= stringToTest,
		Message 	:= 'the assertion changed $'stringToTest$''
	);
	
CNM_AssertionInterfaces.UnicodeStringLengthUnit.CHARACTERS_NFD:	
	currentStringLengthUnit := 'NFD';
	
	CNM_UnicodeUtilities.NormalizeUtf8String(
		utf8StringBuffer := ADR(stringToTest),
		normalForm := CNM_UnicodeUtilities.NormalizationForm.NFD,
		normalizedStringBuffer := ADR(normalizedStringToTest),
		bufferSize := Tc2_System.MAX_STRING_LENGTH + 1,
		normalizedStringLength => normalizedLength
	);
	CNM_UnicodeUtilities.GetUtf8StringLength(
		stringAddress := ADR(normalizedStringToTest),
		characterCount => stringToTestCodePointCount
	);
		
	assertionIsWrong := stringToTestCodePointCount <> expectedLength;
	
	message := SEL(
		assertionIsWrong,
		'stringToCheck is $'%s$' with expectedLength %u assertion must be TRUE  (%S)', 
		'stringToCheck is $'%s$' with expectedLength %u assertion must be FALSE  (%S)'
	);
	
	messageStringBuilder(
		sFormat := message,
		arg1 := THIS^.AnyToArg(stringToTestAsString),
		arg2 := THIS^.AnyToArg(expectedLength),
		arg3 := THIS^.AnyToArg(currentStringLengthUnit)
	);
	
	THIS^.assertorContainer.assertor.assert.strings.unicode.lengthIsExact(
		stringToCheck := stringToTest,
		expectedLength := expectedLength,
		stringLengthUnit := CNM_AssertionInterfaces.UnicodeStringLengthUnit.CHARACTERS_NFD,
		message			:= ''
	);
	
	THIS^.AssertEquals_BOOL(
		Expected 	:= assertionIsWrong,
		Actual 		:= THIS^.assertorContainer.wasAssertionWrong,
		Message 	:= messageStringBuilder.sOut
	);
	
	THIS^.AssertEquals_STRING(
		Expected 	:= stringToTestBeforeAssertion,
		Actual 		:= stringToTest,
		Message 	:= 'the assertion changed $'stringToTest$''
	);
	
CNM_AssertionInterfaces.UnicodeStringLengthUnit.CHARACTERS_NFC:	
	currentStringLengthUnit := 'NFC';
	
	CNM_UnicodeUtilities.NormalizeUtf8String(
		utf8StringBuffer := ADR(stringToTest),
		normalForm := CNM_UnicodeUtilities.NormalizationForm.NFC,
		normalizedStringBuffer := ADR(normalizedStringToTest),
		bufferSize := Tc2_System.MAX_STRING_LENGTH + 1,
		normalizedStringLength => normalizedLength
	);
	CNM_UnicodeUtilities.GetUtf8StringLength(
		stringAddress := ADR(normalizedStringToTest),
		characterCount => stringToTestCodePointCount
	);
		
	assertionIsWrong := stringToTestCodePointCount <> expectedLength;
	
	message := SEL(
		assertionIsWrong,
		'stringToCheck is $'%s$' with expectedLength %u assertion must be TRUE  (%S)', 
		'stringToCheck is $'%s$' with expectedLength %u assertion must be FALSE  (%S)'
	);
	
	messageStringBuilder(
		sFormat := message,
		arg1 := THIS^.AnyToArg(stringToTestAsString),
		arg2 := THIS^.AnyToArg(expectedLength),
		arg3 := THIS^.AnyToArg(currentStringLengthUnit)
	);
	
	THIS^.assertorContainer.assertor.assert.strings.unicode.lengthIsExact(
		stringToCheck := stringToTest,
		expectedLength := expectedLength,
		stringLengthUnit := CNM_AssertionInterfaces.UnicodeStringLengthUnit.CHARACTERS_NFC,
		message			:= ''
	);
	
	THIS^.AssertEquals_BOOL(
		Expected 	:= assertionIsWrong,
		Actual 		:= THIS^.assertorContainer.wasAssertionWrong,
		Message 	:= messageStringBuilder.sOut
	);
	
	THIS^.AssertEquals_STRING(
		Expected 	:= stringToTestBeforeAssertion,
		Actual 		:= stringToTest,
		Message 	:= 'the assertion changed $'stringToTest$''
	);
	
CNM_AssertionInterfaces.UnicodeStringLengthUnit.VISIBLE_CHARACTERS:	
	currentStringLengthUnit := 'VISIBLE_CHARACTERS';
	
	assertionIsWrong := stringToTestVisibleCharacters <> expectedLength;
	
	message := SEL(
		assertionIsWrong,
		'stringToCheck is $'%s$' with expectedLength %u assertion must be TRUE  (%S)', 
		'stringToCheck is $'%s$' with expectedLength %u assertion must be FALSE  (%S)'
	);
	
	messageStringBuilder(
		sFormat := message,
		arg1 := THIS^.AnyToArg(stringToTestAsString),
		arg2 := THIS^.AnyToArg(expectedLength),
		arg3 := THIS^.AnyToArg(currentStringLengthUnit)
	);
	
	THIS^.assertorContainer.assertor.assert.strings.unicode.lengthIsExact(
		stringToCheck := stringToTest,
		expectedLength := expectedLength,
		stringLengthUnit := CNM_AssertionInterfaces.UnicodeStringLengthUnit.VISIBLE_CHARACTERS,
		message			:= ''
	);
	
	THIS^.AssertEquals_BOOL(
		Expected 	:= assertionIsWrong,
		Actual 		:= THIS^.assertorContainer.wasAssertionWrong,
		Message 	:= messageStringBuilder.sOut
	);
	
	THIS^.AssertEquals_STRING(
		Expected 	:= stringToTestBeforeAssertion,
		Actual 		:= stringToTest,
		Message 	:= 'the assertion changed $'stringToTest$''
	);
	
CNM_AssertionInterfaces.UnicodeStringLengthUnit.WIDTH:	
	currentStringLengthUnit := 'WIDTH';
	
	assertionIsWrong := TO_UDINT(stringToTestWidth) <> expectedLength;
	
	message := SEL(
		assertionIsWrong,
		'stringToCheck is $'%s$' with expectedLength %u assertion must be TRUE  (%S)', 
		'stringToCheck is $'%s$' with expectedLength %u assertion must be FALSE  (%S)'
	);
	
	messageStringBuilder(
		sFormat := message,
		arg1 := THIS^.AnyToArg(stringToTestAsString),
		arg2 := THIS^.AnyToArg(expectedLength),
		arg3 := THIS^.AnyToArg(currentStringLengthUnit)
	);
	
	THIS^.assertorContainer.assertor.assert.strings.unicode.lengthIsExact(
		stringToCheck := stringToTest,
		expectedLength := expectedLength,
		stringLengthUnit := CNM_AssertionInterfaces.UnicodeStringLengthUnit.WIDTH,
		message			:= ''
	);
	
	THIS^.AssertEquals_BOOL(
		Expected 	:= assertionIsWrong,
		Actual 		:= THIS^.assertorContainer.wasAssertionWrong,
		Message 	:= messageStringBuilder.sOut
	);

	THIS^.AssertEquals_STRING(
		Expected 	:= stringToTestBeforeAssertion,
		Actual 		:= stringToTest,
		Message 	:= 'the assertion changed $'stringToTest$''
	);

END_CASE
END_METHOD

(*
short summary
==================
This test method tests ``assert.string.unicode.lengthIsMax``
method of CNM_AssertionInterfaces library with various inputs

.. <legal notes>

legal notes
=================
| SPDX-FileCopyrightText: © 2022 ekvip automation GmbH <info@ekvip.de>
| SPDX-License-Identifier: Apache-2.0
| For details check: Apache-2.0_

.. _Apache-2.0: https://www.apache.org/licenses/LICENSE-2.0

.. </legal notes>

*)


METHOD testLengthIsMax : BOOL
VAR_INPUT
	(* for the test it's the parameter ``stringToCheck`` *)
	{attribute 'TcEncoding' := 'UTF-8'}
	stringToTest 			:Tc2_System.T_MaxString;
	(* for the test it's the parameter ``maxLength`` *)
	expectedLength			:UDINT;
	(* UnicodeStringLengthUnit the input is tested for *)
	stringLengthUnit		:CNM_AssertionInterfaces.UnicodeStringLengthUnit;
	(* contains ``stringToTest`` in only ascii charachters for test output *)
	stringToTestPrintable	:Tc2_System.T_MaxString := '';
END_VAR
VAR 
	(* just the expectation if the assertion to test must be worng or true *)
	assertionIsWrong				:BOOL;
	(* contains the format string for the test message *)
	message							:Tc2_System.T_MaxString;
	(* used for placeholder string if stringToTest can't be printed *)
	stringToTestAsString 			:Tc2_System.T_MaxString;
	(* holds string with current ´´stringLengthUnit´´ for the test message*)
	currentStringLengthUnit 		:Tc2_System.T_MaxString;
	(* TwinCAT printf with the test message *)
	messageStringBuilder			:Tc2_Utilities.FB_FormatString;
	(* length of current string to check in bytes *)
	stringToTestByteCount			:UDINT;
	(* length of current string to check in characters *)
	stringToTestCodePointCount		:UDINT;
	(* length of ´´stringToCheck´´ *)
	normalizedLength 				:UDINT;
	(* holds the normalized ´´stringToCheck´´ *)
	{attribute 'TcEncoding' := 'UTF-8'}
	normalizedStringToTest 			:Tc2_System.T_MaxString;
	(* width of ´´stringToCheck´´ *)
	stringToTestWidth 				:DINT;
	(* visible characters of ´´stringToCheck´´ *)
	stringToTestVisibleCharacters	:UDINT := 0;
	(* hold stringToCheck before assertion *)
	stringToTestBeforeAssertion		:Tc2_System.T_MaxString;
END_VAR
THIS^.assertorContainer.resetAssertor();

stringToTestBeforeAssertion := stringToTest;
stringToTestAsString := stringToTest;

CNM_UnicodeUtilities.GetUtf8StringLength(ADR(stringToTest), byteCount => stringToTestByteCount, characterCount => stringToTestCodePointCount,);
CNM_UnicodeUtilities.GetUtf8StringWidth(ADR(stringToTest), visibleCharacters => stringToTestVisibleCharacters, width => stringToTestWidth);

IF (
		Tc2_Standard.LEN(stringToTest) = TO_UINT(Tc2_System.MAX_STRING_LENGTH)
) THEN
	stringToTestAsString := 'String with Tc2_System.MAX_STRING_LENGTH characters';
END_IF
IF (
		LEN(stringToTestPrintable) <> 0
) THEN
	stringToTestAsString := stringToTestPrintable;
END_IF

CASE stringLengthUnit OF
	
CNM_AssertionInterfaces.UnicodeStringLengthUnit.BYTES:
	currentStringLengthUnit := 'BYTES';
	
	assertionIsWrong := stringToTestByteCount > expectedLength;
	
	message := SEL(
		assertionIsWrong,
		'stringToCheck is $'%s$' with expectedLength %u assertion must be TRUE  (%S)', 
		'stringToCheck is $'%s$' with expectedLength %u assertion must be FALSE  (%S)'
	);
	
	messageStringBuilder(
		sFormat := message,
		arg1 := THIS^.AnyToArg(stringToTestAsString),
		arg2 := THIS^.AnyToArg(expectedLength),
		arg3 := THIS^.AnyToArg(currentStringLengthUnit)
	);
	
	THIS^.assertorContainer.assertor.assert.strings.unicode.lengthIsMax(
		stringToCheck := stringToTest,
		maxLength := expectedLength,
		stringLengthUnit := CNM_AssertionInterfaces.UnicodeStringLengthUnit.BYTES,
		message			:= ''
	);
	
	THIS^.AssertEquals_BOOL(
		Expected 	:= assertionIsWrong,
		Actual 		:= THIS^.assertorContainer.wasAssertionWrong,
		Message 	:= messageStringBuilder.sOut
	);
	
	THIS^.AssertEquals_STRING(
		Expected 	:= stringToTestBeforeAssertion,
		Actual 		:= stringToTest,
		Message 	:= 'the assertion changed $'stringToTest$''
	);
	
CNM_AssertionInterfaces.UnicodeStringLengthUnit.CHARACTERS:	
	currentStringLengthUnit := 'CHARACTERS';
	THIS^.assertorContainer.resetAssertor();
	
	assertionIsWrong := stringToTestCodePointCount > expectedLength;
	
	message := SEL(
		assertionIsWrong,
		'stringToCheck is $'%s$' with expectedLength %u assertion must be TRUE  (%S)', 
		'stringToCheck is $'%s$' with expectedLength %u assertion must be FALSE  (%S)'
	);
	
	messageStringBuilder(
		sFormat := message,
		arg1 := THIS^.AnyToArg(stringToTestAsString),
		arg2 := THIS^.AnyToArg(expectedLength),
		arg3 := THIS^.AnyToArg(currentStringLengthUnit)
	);
	
	THIS^.assertorContainer.assertor.assert.strings.unicode.lengthIsMax(
		stringToCheck := stringToTest,
		maxLength := expectedLength,
		stringLengthUnit := CNM_AssertionInterfaces.UnicodeStringLengthUnit.CHARACTERS,
		message			:= ''
	);
	
	THIS^.AssertEquals_BOOL(
		Expected 	:= assertionIsWrong,
		Actual 		:= THIS^.assertorContainer.wasAssertionWrong,
		Message 	:= messageStringBuilder.sOut
	);
	
	THIS^.AssertEquals_STRING(
		Expected 	:= stringToTestBeforeAssertion,
		Actual 		:= stringToTest,
		Message 	:= 'the assertion changed $'stringToTest$''
	);
	
CNM_AssertionInterfaces.UnicodeStringLengthUnit.CHARACTERS_NFD:	
	currentStringLengthUnit := 'NFD';
	THIS^.assertorContainer.resetAssertor();
	
	CNM_UnicodeUtilities.NormalizeUtf8String(
		utf8StringBuffer := ADR(stringToTest),
		normalForm := CNM_UnicodeUtilities.NormalizationForm.NFD,
		normalizedStringBuffer := ADR(normalizedStringToTest),
		bufferSize := Tc2_System.MAX_STRING_LENGTH + 1,
		normalizedStringLength => normalizedLength
	);
	CNM_UnicodeUtilities.GetUtf8StringLength(
		stringAddress := ADR(normalizedStringToTest),
		characterCount => stringToTestCodePointCount
	);
		
	assertionIsWrong := stringToTestCodePointCount > expectedLength;
	
	message := SEL(
		assertionIsWrong,
		'stringToCheck is $'%s$' with expectedLength %u assertion must be TRUE  (%S)', 
		'stringToCheck is $'%s$' with expectedLength %u assertion must be FALSE  (%S)'
	);
	
	messageStringBuilder(
		sFormat := message,
		arg1 := THIS^.AnyToArg(stringToTestAsString),
		arg2 := THIS^.AnyToArg(expectedLength),
		arg3 := THIS^.AnyToArg(currentStringLengthUnit)
	);
	
	THIS^.assertorContainer.assertor.assert.strings.unicode.lengthIsMax(
		stringToCheck := stringToTest,
		maxLength := expectedLength,
		stringLengthUnit := CNM_AssertionInterfaces.UnicodeStringLengthUnit.CHARACTERS_NFD,
		message			:= ''
	);
	
	THIS^.AssertEquals_BOOL(
		Expected 	:= assertionIsWrong,
		Actual 		:= THIS^.assertorContainer.wasAssertionWrong,
		Message 	:= messageStringBuilder.sOut
	);
	
	THIS^.AssertEquals_STRING(
		Expected 	:= stringToTestBeforeAssertion,
		Actual 		:= stringToTest,
		Message 	:= 'the assertion changed $'stringToTest$''
	);
	
CNM_AssertionInterfaces.UnicodeStringLengthUnit.CHARACTERS_NFC:	
	currentStringLengthUnit := 'NFC';
	THIS^.assertorContainer.resetAssertor();
	
	CNM_UnicodeUtilities.NormalizeUtf8String(
		utf8StringBuffer := ADR(stringToTest),
		normalForm := CNM_UnicodeUtilities.NormalizationForm.NFC,
		normalizedStringBuffer := ADR(normalizedStringToTest),
		bufferSize := Tc2_System.MAX_STRING_LENGTH + 1,
		normalizedStringLength => normalizedLength
	);
	CNM_UnicodeUtilities.GetUtf8StringLength(
		stringAddress := ADR(normalizedStringToTest),
		characterCount => stringToTestCodePointCount
	);
		
	assertionIsWrong := stringToTestCodePointCount > expectedLength;
	
	message := SEL(
		assertionIsWrong,
		'stringToCheck is $'%s$' with expectedLength %u assertion must be TRUE  (%S)', 
		'stringToCheck is $'%s$' with expectedLength %u assertion must be FALSE  (%S)'
	);
	
	messageStringBuilder(
		sFormat := message,
		arg1 := THIS^.AnyToArg(stringToTestAsString),
		arg2 := THIS^.AnyToArg(expectedLength),
		arg3 := THIS^.AnyToArg(currentStringLengthUnit)
	);
	
	THIS^.assertorContainer.assertor.assert.strings.unicode.lengthIsMax(
		stringToCheck := stringToTest,
		maxLength := expectedLength,
		stringLengthUnit := CNM_AssertionInterfaces.UnicodeStringLengthUnit.CHARACTERS_NFC,
		message			:= ''
	);
	
	THIS^.AssertEquals_BOOL(
		Expected 	:= assertionIsWrong,
		Actual 		:= THIS^.assertorContainer.wasAssertionWrong,
		Message 	:= messageStringBuilder.sOut
	);
	
	THIS^.AssertEquals_STRING(
		Expected 	:= stringToTestBeforeAssertion,
		Actual 		:= stringToTest,
		Message 	:= 'the assertion changed $'stringToTest$''
	);
	
CNM_AssertionInterfaces.UnicodeStringLengthUnit.VISIBLE_CHARACTERS:	
	currentStringLengthUnit := 'VISIBLE_CHARACTERS';
	THIS^.assertorContainer.resetAssertor();
	
	assertionIsWrong := stringToTestVisibleCharacters > expectedLength;
	
	message := SEL(
		assertionIsWrong,
		'stringToCheck is $'%s$' with expectedLength %u assertion must be TRUE  (%S)', 
		'stringToCheck is $'%s$' with expectedLength %u assertion must be FALSE  (%S)'
	);
	
	messageStringBuilder(
		sFormat := message,
		arg1 := THIS^.AnyToArg(stringToTestAsString),
		arg2 := THIS^.AnyToArg(expectedLength),
		arg3 := THIS^.AnyToArg(currentStringLengthUnit)
	);
	
	THIS^.assertorContainer.assertor.assert.strings.unicode.lengthIsMax(
		stringToCheck := stringToTest,
		maxLength := expectedLength,
		stringLengthUnit := CNM_AssertionInterfaces.UnicodeStringLengthUnit.VISIBLE_CHARACTERS,
		message			:= ''
	);
	
	THIS^.AssertEquals_BOOL(
		Expected 	:= assertionIsWrong,
		Actual 		:= THIS^.assertorContainer.wasAssertionWrong,
		Message 	:= messageStringBuilder.sOut
	);
	
	THIS^.AssertEquals_STRING(
		Expected 	:= stringToTestBeforeAssertion,
		Actual 		:= stringToTest,
		Message 	:= 'the assertion changed $'stringToTest$''
	);
	
CNM_AssertionInterfaces.UnicodeStringLengthUnit.WIDTH:	
	currentStringLengthUnit := 'WIDTH';
	THIS^.assertorContainer.resetAssertor();
	
	assertionIsWrong := TO_UDINT(stringToTestWidth) > expectedLength;
	
	message := SEL(
		assertionIsWrong,
		'stringToCheck is $'%s$' with expectedLength %u assertion must be TRUE  (%S)', 
		'stringToCheck is $'%s$' with expectedLength %u assertion must be FALSE  (%S)'
	);
	
	messageStringBuilder(
		sFormat := message,
		arg1 := THIS^.AnyToArg(stringToTestAsString),
		arg2 := THIS^.AnyToArg(expectedLength),
		arg3 := THIS^.AnyToArg(currentStringLengthUnit)
	);
	
	THIS^.assertorContainer.assertor.assert.strings.unicode.lengthIsMax(
		stringToCheck := stringToTest,
		maxLength := expectedLength,
		stringLengthUnit := CNM_AssertionInterfaces.UnicodeStringLengthUnit.WIDTH,
		message			:= ''
	);
	
	THIS^.AssertEquals_BOOL(
		Expected 	:= assertionIsWrong,
		Actual 		:= THIS^.assertorContainer.wasAssertionWrong,
		Message 	:= messageStringBuilder.sOut
	);

	THIS^.AssertEquals_STRING(
		Expected 	:= stringToTestBeforeAssertion,
		Actual 		:= stringToTest,
		Message 	:= 'the assertion changed $'stringToTest$''
	);

END_CASE
END_METHOD

(*
short summary
==================
This test method tests ``assert.string.unicode.lengthIsMin``
method of CNM_AssertionInterfaces library with various inputs

.. <legal notes>

legal notes
=================
| SPDX-FileCopyrightText: © 2022 ekvip automation GmbH <info@ekvip.de>
| SPDX-License-Identifier: Apache-2.0
| For details check: Apache-2.0_

.. _Apache-2.0: https://www.apache.org/licenses/LICENSE-2.0

.. </legal notes>

*)


METHOD testLengthIsMin : BOOL
VAR_INPUT
	(* for the test it's the parameter ``stringToCheck`` *)
	{attribute 'TcEncoding' := 'UTF-8'}
	stringToTest 			:Tc2_System.T_MaxString;
	(* for the test it's the parameter ``minLength`` *)
	expectedLength 			:UDINT;
	(* UnicodeStringLengthUnit the input is tested for *)
	stringLengthUnit		:CNM_AssertionInterfaces.UnicodeStringLengthUnit;
	(* contains ``stringToTest`` in only ascii charachters for test output *)
	stringToTestPrintable	:Tc2_System.T_MaxString := '';
END_VAR
VAR 
	(* just the expectation if the assertion to test must be worng or true *)
	assertionIsWrong				:BOOL;
	(* contains the format string for the test message *)
	message							:Tc2_System.T_MaxString;
	(* used for placeholder string if stringToTest can't be printed *)
	stringToTestAsString 			:Tc2_System.T_MaxString;
	(* holds string with current ´´stringLengthUnit´´ for the test message*)
	currentStringLengthUnit 		:Tc2_System.T_MaxString;
	(* TwinCAT printf with the test message *)
	messageStringBuilder			:Tc2_Utilities.FB_FormatString;
	(* length of current string to check in bytes *)
	stringToTestByteCount			:UDINT;
	(* length of current string to check in characters *)
	stringToTestCodePointCount		:UDINT;
	(* length of ´´stringToCheck´´ *)
	normalizedLength 				:UDINT;
	(* holds the normalized ´´stringToCheck´´ *)
	{attribute 'TcEncoding' := 'UTF-8'}
	normalizedStringToTest 			:Tc2_System.T_MaxString;
	(* width of ´´stringToCheck´´ *)
	stringToTestWidth 				:DINT;
	(* visible characters of ´´stringToCheck´´ *)
	stringToTestVisibleCharacters	:UDINT := 0;
	(* hold stringToCheck before assertion *)
	stringToTestBeforeAssertion		:Tc2_System.T_MaxString;
END_VAR
THIS^.assertorContainer.resetAssertor();

stringToTestBeforeAssertion := stringToTest;
stringToTestAsString := stringToTest;

CNM_UnicodeUtilities.GetUtf8StringLength(ADR(stringToTest), byteCount => stringToTestByteCount, characterCount => stringToTestCodePointCount,);
CNM_UnicodeUtilities.GetUtf8StringWidth(ADR(stringToTest), visibleCharacters => stringToTestVisibleCharacters, width => stringToTestWidth);

IF (
		Tc2_Standard.LEN(stringToTest) = TO_UINT(Tc2_System.MAX_STRING_LENGTH)
) THEN
	stringToTestAsString := 'String with Tc2_System.MAX_STRING_LENGTH characters';
END_IF
IF (
		LEN(stringToTestPrintable) <> 0
) THEN
	stringToTestAsString := stringToTestPrintable;
END_IF

CASE stringLengthUnit OF
	
CNM_AssertionInterfaces.UnicodeStringLengthUnit.BYTES:
	currentStringLengthUnit := 'BYTES';
	
	assertionIsWrong := stringToTestByteCount < expectedLength;
	
	message := SEL(
		assertionIsWrong,
		'stringToCheck is $'%s$' with expectedLength %u assertion must be TRUE  (%S)', 
		'stringToCheck is $'%s$' with expectedLength %u assertion must be FALSE  (%S)'
	);
	
	messageStringBuilder(
		sFormat := message,
		arg1 := THIS^.AnyToArg(stringToTestAsString),
		arg2 := THIS^.AnyToArg(expectedLength),
		arg3 := THIS^.AnyToArg(currentStringLengthUnit)
	);
	
	THIS^.assertorContainer.assertor.assert.strings.unicode.lengthIsMin(
		stringToCheck := stringToTest,
		minLength := expectedLength,
		stringLengthUnit := CNM_AssertionInterfaces.UnicodeStringLengthUnit.BYTES,
		message			:= ''
	);
	
	THIS^.AssertEquals_BOOL(
		Expected 	:= assertionIsWrong,
		Actual 		:= THIS^.assertorContainer.wasAssertionWrong,
		Message 	:= messageStringBuilder.sOut
	);
	
	THIS^.AssertEquals_STRING(
		Expected 	:= stringToTestBeforeAssertion,
		Actual 		:= stringToTest,
		Message 	:= 'the assertion changed $'stringToTest$''
	);
	
CNM_AssertionInterfaces.UnicodeStringLengthUnit.CHARACTERS:	
	currentStringLengthUnit := 'CHARACTERS';
	THIS^.assertorContainer.resetAssertor();
	
	assertionIsWrong := stringToTestCodePointCount < expectedLength;
	
	message := SEL(
		assertionIsWrong,
		'stringToCheck is $'%s$' with expectedLength %u assertion must be TRUE  (%S)', 
		'stringToCheck is $'%s$' with expectedLength %u assertion must be FALSE  (%S)'
	);
	
	messageStringBuilder(
		sFormat := message,
		arg1 := THIS^.AnyToArg(stringToTestAsString),
		arg2 := THIS^.AnyToArg(expectedLength),
		arg3 := THIS^.AnyToArg(currentStringLengthUnit)
	);
	
	THIS^.assertorContainer.assertor.assert.strings.unicode.lengthIsMin(
		stringToCheck := stringToTest,
		minLength := expectedLength,
		stringLengthUnit := CNM_AssertionInterfaces.UnicodeStringLengthUnit.CHARACTERS,
		message			:= ''
	);
	
	THIS^.AssertEquals_BOOL(
		Expected 	:= assertionIsWrong,
		Actual 		:= THIS^.assertorContainer.wasAssertionWrong,
		Message 	:= messageStringBuilder.sOut
	);
	
	THIS^.AssertEquals_STRING(
		Expected 	:= stringToTestBeforeAssertion,
		Actual 		:= stringToTest,
		Message 	:= 'the assertion changed $'stringToTest$''
	);
	
CNM_AssertionInterfaces.UnicodeStringLengthUnit.CHARACTERS_NFD:	
	currentStringLengthUnit := 'NFD';
	THIS^.assertorContainer.resetAssertor();
	
	CNM_UnicodeUtilities.NormalizeUtf8String(
		utf8StringBuffer := ADR(stringToTest),
		normalForm := CNM_UnicodeUtilities.NormalizationForm.NFD,
		normalizedStringBuffer := ADR(normalizedStringToTest),
		bufferSize := Tc2_System.MAX_STRING_LENGTH + 1,
		normalizedStringLength => normalizedLength
	);
	CNM_UnicodeUtilities.GetUtf8StringLength(
		stringAddress := ADR(normalizedStringToTest),
		characterCount => stringToTestCodePointCount
	);
		
	assertionIsWrong := stringToTestCodePointCount < expectedLength;
	
	message := SEL(
		assertionIsWrong,
		'stringToCheck is $'%s$' with expectedLength %u assertion must be TRUE  (%S)', 
		'stringToCheck is $'%s$' with expectedLength %u assertion must be FALSE  (%S)'
	);
	
	messageStringBuilder(
		sFormat := message,
		arg1 := THIS^.AnyToArg(stringToTestAsString),
		arg2 := THIS^.AnyToArg(expectedLength),
		arg3 := THIS^.AnyToArg(currentStringLengthUnit)
	);
	
	THIS^.assertorContainer.assertor.assert.strings.unicode.lengthIsMin(
		stringToCheck := stringToTest,
		minLength := expectedLength,
		stringLengthUnit := CNM_AssertionInterfaces.UnicodeStringLengthUnit.CHARACTERS_NFD,
		message			:= ''
	);
	
	THIS^.AssertEquals_BOOL(
		Expected 	:= assertionIsWrong,
		Actual 		:= THIS^.assertorContainer.wasAssertionWrong,
		Message 	:= messageStringBuilder.sOut
	);
	
	THIS^.AssertEquals_STRING(
		Expected 	:= stringToTestBeforeAssertion,
		Actual 		:= stringToTest,
		Message 	:= 'the assertion changed $'stringToTest$''
	);
	
CNM_AssertionInterfaces.UnicodeStringLengthUnit.CHARACTERS_NFC:	
	currentStringLengthUnit := 'NFC';
	THIS^.assertorContainer.resetAssertor();
	
	CNM_UnicodeUtilities.NormalizeUtf8String(
		utf8StringBuffer := ADR(stringToTest),
		normalForm := CNM_UnicodeUtilities.NormalizationForm.NFC,
		normalizedStringBuffer := ADR(normalizedStringToTest),
		bufferSize := Tc2_System.MAX_STRING_LENGTH + 1,
		normalizedStringLength => normalizedLength
	);
	CNM_UnicodeUtilities.GetUtf8StringLength(
		stringAddress := ADR(normalizedStringToTest),
		characterCount => stringToTestCodePointCount
	);
		
	assertionIsWrong := stringToTestCodePointCount < expectedLength;
	
	message := SEL(
		assertionIsWrong,
		'stringToCheck is $'%s$' with expectedLength %u assertion must be TRUE  (%S)', 
		'stringToCheck is $'%s$' with expectedLength %u assertion must be FALSE  (%S)'
	);
	
	messageStringBuilder(
		sFormat := message,
		arg1 := THIS^.AnyToArg(stringToTestAsString),
		arg2 := THIS^.AnyToArg(expectedLength),
		arg3 := THIS^.AnyToArg(currentStringLengthUnit)
	);
	
	THIS^.assertorContainer.assertor.assert.strings.unicode.lengthIsMin(
		stringToCheck := stringToTest,
		minLength := expectedLength,
		stringLengthUnit := CNM_AssertionInterfaces.UnicodeStringLengthUnit.CHARACTERS_NFC,
		message			:= ''
	);
	
	THIS^.AssertEquals_BOOL(
		Expected 	:= assertionIsWrong,
		Actual 		:= THIS^.assertorContainer.wasAssertionWrong,
		Message 	:= messageStringBuilder.sOut
	);
	
	THIS^.AssertEquals_STRING(
		Expected 	:= stringToTestBeforeAssertion,
		Actual 		:= stringToTest,
		Message 	:= 'the assertion changed $'stringToTest$''
	);
	
CNM_AssertionInterfaces.UnicodeStringLengthUnit.VISIBLE_CHARACTERS:	
	currentStringLengthUnit := 'VISIBLE_CHARACTERS';
	THIS^.assertorContainer.resetAssertor();
	
	assertionIsWrong := stringToTestVisibleCharacters < expectedLength;
	
	message := SEL(
		assertionIsWrong,
		'stringToCheck is $'%s$' with expectedLength %u assertion must be TRUE  (%S)', 
		'stringToCheck is $'%s$' with expectedLength %u assertion must be FALSE  (%S)'
	);
	
	messageStringBuilder(
		sFormat := message,
		arg1 := THIS^.AnyToArg(stringToTestAsString),
		arg2 := THIS^.AnyToArg(expectedLength),
		arg3 := THIS^.AnyToArg(currentStringLengthUnit)
	);
	
	THIS^.assertorContainer.assertor.assert.strings.unicode.lengthIsMin(
		stringToCheck := stringToTest,
		minLength := expectedLength,
		stringLengthUnit := CNM_AssertionInterfaces.UnicodeStringLengthUnit.VISIBLE_CHARACTERS,
		message			:= ''
	);
	
	THIS^.AssertEquals_BOOL(
		Expected 	:= assertionIsWrong,
		Actual 		:= THIS^.assertorContainer.wasAssertionWrong,
		Message 	:= messageStringBuilder.sOut
	);
	
	THIS^.AssertEquals_STRING(
		Expected 	:= stringToTestBeforeAssertion,
		Actual 		:= stringToTest,
		Message 	:= 'the assertion changed $'stringToTest$''
	);
	
CNM_AssertionInterfaces.UnicodeStringLengthUnit.WIDTH:	
	currentStringLengthUnit := 'WIDTH';
	THIS^.assertorContainer.resetAssertor();
	
	assertionIsWrong := TO_UDINT(stringToTestWidth) < expectedLength;
	
	message := SEL(
		assertionIsWrong,
		'stringToCheck is $'%s$' with expectedLength %u assertion must be TRUE  (%S)', 
		'stringToCheck is $'%s$' with expectedLength %u assertion must be FALSE  (%S)'
	);
	
	messageStringBuilder(
		sFormat := message,
		arg1 := THIS^.AnyToArg(stringToTestAsString),
		arg2 := THIS^.AnyToArg(expectedLength),
		arg3 := THIS^.AnyToArg(currentStringLengthUnit)
	);
	
	THIS^.assertorContainer.assertor.assert.strings.unicode.lengthIsMin(
		stringToCheck := stringToTest,
		minLength := expectedLength,
		stringLengthUnit := CNM_AssertionInterfaces.UnicodeStringLengthUnit.WIDTH,
		message			:= ''
	);
	
	THIS^.AssertEquals_BOOL(
		Expected 	:= assertionIsWrong,
		Actual 		:= THIS^.assertorContainer.wasAssertionWrong,
		Message 	:= messageStringBuilder.sOut
	);
	
	THIS^.AssertEquals_STRING(
		Expected 	:= stringToTestBeforeAssertion,
		Actual 		:= stringToTest,
		Message 	:= 'the assertion changed $'stringToTest$''
	);
	
END_CASE
END_METHOD

(*
short summary
==================
This test method tests ``assert.string.unicode.startsWith``
method of CNM_AssertionInterfaces library with various inputs

.. <legal notes>

legal notes
=================
| SPDX-FileCopyrightText: © 2022 ekvip automation GmbH <info@ekvip.de>
| SPDX-License-Identifier: Apache-2.0
| For details check: Apache-2.0_

.. _Apache-2.0: https://www.apache.org/licenses/LICENSE-2.0

.. </legal notes>

*)


METHOD testStartsWith : BOOL
VAR_INPUT
	(* for the test it's the parameter ``stringToCheck`` *)
	{attribute 'TcEncoding' := 'UTF-8'}
	stringToTest 	:Tc2_System.T_MaxString;
	(* for the test it's the parameter ``end`` *)
	{attribute 'TcEncoding' := 'UTF-8'}
	expectedString 	:Tc2_System.T_MaxString;
END_VAR
VAR 
	(* just the expectation if the assertion to test must be worng or true *)
	assertionIsWrong				:BOOL;
	(* contains the format string for the test message *)
	message							:Tc2_System.T_MaxString;
	(* used for placeholder string if stringToTest can't be printed *)
	stringToTestAsString 			:Tc2_System.T_MaxString;
	(* used for placeholder string if expectedString can't be printed *)
	expectedStringAsString 			:Tc2_System.T_MaxString;
	(* contains stringToTest in normalized form *)
	normalizedStringToTest			:Tc2_System.T_MaxString;
	(* contains expectedString in normalized form *)
	normalizedExpectedString		:Tc2_System.T_MaxString;
	(* holds characterCount of ``expectedString`` *)
	expectedCharacterCount			:UDINT;
	(* TwinCAT printf with the test message *)
	messageStringBuilder			:Tc2_Utilities.FB_FormatString;
	(* hold stringToCheck before assertion *)
	stringToTestBeforeAssertion		:Tc2_System.T_MaxString;
	(* hold expectedString before assertion *)
	expectedStringBeforeAssertion	:Tc2_System.T_MaxString;
END_VAR
THIS^.assertorContainer.resetAssertor();

stringToTestBeforeAssertion := stringToTest;
expectedStringBeforeAssertion := expectedString;
stringToTestAsString := stringToTest;
expectedStringAsString := expectedString;

CNM_UnicodeUtilities.GetUtf8StringLength(
	ADR(expectedString),
	characterCount => expectedCharacterCount
);
assertionIsWrong := ((
		CNM_UnicodeUtilities.FindInUtf8String(
			ADR(stringToTest),
			ADR(expectedString),
		) <> 1
	) AND (
		expectedCharacterCount <> 0
	)
);

message := SEL(
	assertionIsWrong,
	'stringToCheck is $'%s$' start is $'%s$' assertion must be TRUE', 
	'stringToCheck is $'%s$' start is $'%s$' assertion must be FALSE'
);

IF (
		Tc2_Standard.LEN(stringToTest) = TO_UINT(Tc2_System.MAX_STRING_LENGTH)
) THEN
	stringToTestAsString := 'String with Tc2_System.MAX_STRING_LENGTH characters';
END_IF
IF (
		Tc2_Standard.LEN(expectedString) = TO_UINT(Tc2_System.MAX_STRING_LENGTH)
) THEN
	expectedStringAsString := 'String with Tc2_System.MAX_STRING_LENGTH characters';
END_IF

messageStringBuilder(
	sFormat := message,
	arg1 := THIS^.AnyToArg(stringToTestAsString),
	arg2 := THIS^.AnyToArg(expectedStringAsString)
);


THIS^.assertorContainer.assertor.assert.strings.unicode.startsWith(
	stringToCheck := stringToTest,
	start := expectedString,
	ignoreCases := FALSE,
	trim := FALSE,
	normalizeStrings := FALSE,
	message			:= ''
);

THIS^.AssertEquals_BOOL(
	Expected 	:= assertionIsWrong,
	Actual 		:= THIS^.assertorContainer.wasAssertionWrong,
	Message 	:= messageStringBuilder.sOut
);

THIS^.AssertEquals_STRING(
	Expected 	:= stringToTestBeforeAssertion,
	Actual 		:= stringToTest,
	Message 	:= 'the assertion changed $'stringToTest$''
);

THIS^.AssertEquals_STRING(
	Expected 	:= expectedStringBeforeAssertion,
	Actual 		:= expectedString,
	Message 	:= 'the assertion changed $'expectedString$''
);

THIS^.assertorContainer.resetAssertor();

CNM_UnicodeUtilities.NormalizeUtf8String(
	utf8StringBuffer := ADR(stringToTest),
	bufferSize := Tc2_System.MAX_STRING_LENGTH + 1,
	normalizedStringBuffer := ADR(normalizedStringToTest),
	normalForm := CNM_UnicodeUtilities.NormalizationForm.NFD
);
CNM_UnicodeUtilities.NormalizeUtf8String(
	utf8StringBuffer := ADR(expectedString),
	bufferSize := Tc2_System.MAX_STRING_LENGTH + 1,
	normalizedStringBuffer := ADR(normalizedExpectedString),
	normalForm := CNM_UnicodeUtilities.NormalizationForm.NFD
);

CNM_UnicodeUtilities.GetUtf8StringLength(
	ADR(normalizedExpectedString),
	characterCount => expectedCharacterCount
);
assertionIsWrong := ((
		CNM_UnicodeUtilities.FindInUtf8String(
			ADR(normalizedStringToTest),
			ADR(normalizedExpectedString),
		) <> 1
	) AND (
		expectedCharacterCount <> 0
	)
);

THIS^.assertorContainer.assertor.assert.strings.unicode.startsWith(
	stringToCheck := stringToTest,
	start := expectedString,
	ignoreCases := FALSE,
	trim		:= FALSE,
	normalizeStrings := TRUE,
	message			:= ''
);

THIS^.AssertEquals_BOOL(
	Expected 	:= assertionIsWrong,
	Actual 		:= THIS^.assertorContainer.wasAssertionWrong,
	Message 	:= messageStringBuilder.sOut
);

THIS^.AssertEquals_STRING(
	Expected 	:= stringToTestBeforeAssertion,
	Actual 		:= stringToTest,
	Message 	:= 'the assertion changed $'stringToTest$''
);

THIS^.AssertEquals_STRING(
	Expected 	:= expectedStringBeforeAssertion,
	Actual 		:= expectedString,
	Message 	:= 'the assertion changed $'expectedString$''
);
END_METHOD

(*
short summary
==================
This test method tests ``assert.string.unicode.startsWith``
method of CNM_AssertionInterfaces library with various inputs

.. <legal notes>

legal notes
=================
| SPDX-FileCopyrightText: © 2022 ekvip automation GmbH <info@ekvip.de>
| SPDX-License-Identifier: Apache-2.0
| For details check: Apache-2.0_

.. _Apache-2.0: https://www.apache.org/licenses/LICENSE-2.0

.. </legal notes>

*)


METHOD testStartsWithIgnoreCase : BOOL
VAR_INPUT
	(* for the test it's the parameter ``stringToCheck`` *)
	{attribute 'TcEncoding' := 'UTF-8'}
	stringToTest 	:Tc2_System.T_MaxString;
	(* for the test it's the parameter ``end`` *)
	{attribute 'TcEncoding' := 'UTF-8'}
	expectedString	:Tc2_System.T_MaxString;
END_VAR
VAR 
	(* just the expectation if the assertion to test must be worng or true *)
	assertionIsWrong				:BOOL;
	(* contains the format string for the test message *)
	message							:Tc2_System.T_MaxString;
	(* contains ´´stringToTest´´ in upper case *)
	upperStringToTest				:Tc2_System.T_MaxString;
	(* contains ´´expectedString´´ in upper case *)
	upperExpectedString				:Tc2_System.T_MaxString;
	(* used for placeholder string if stringToTest can't be printed *)
	stringToTestAsString 			:Tc2_System.T_MaxString;
	(* used for placeholder string if expectedString can't be printed *)
	expectedStringAsString 			:Tc2_System.T_MaxString;
	(* contains stringToTest in normalized form *)
	normalizedStringToTest			:Tc2_System.T_MaxString;
	(* contains expectedString in normalized form *)
	normalizedExpectedString		:Tc2_System.T_MaxString;
	(* contains stringToTest in normalized form in upper case*)
	normalizedUpperStringToTest		:Tc2_System.T_MaxString;
	(* contains expectedString in normalized form in upper case*)
	normalizedUpperExpectedString	:Tc2_System.T_MaxString;
	(* holds characterCount of ``expectedString`` *)
	expectedCharacterCount			:UDINT;
	(* TwinCAT printf with the test message *)
	messageStringBuilder			:Tc2_Utilities.FB_FormatString;
	(* hold stringToCheck before assertion *)
	stringToTestBeforeAssertion		:Tc2_System.T_MaxString;
	(* hold expectedString before assertion *)
	expectedStringBeforeAssertion	:Tc2_System.T_MaxString;
END_VAR
THIS^.assertorContainer.resetAssertor();

stringToTestBeforeAssertion := stringToTest;
expectedStringBeforeAssertion := expectedString;
stringToTestAsString := stringToTest;
expectedStringAsString := expectedString;
upperStringToTest := stringToTest;
upperExpectedString := expectedString;

// both Strings to upper case
CNM_UnicodeUtilities.UpperCaseUtf8(ADR(upperStringToTest));
CNM_UnicodeUtilities.UpperCaseUtf8(ADR(upperExpectedString));

CNM_UnicodeUtilities.GetUtf8StringLength(
	ADR(upperExpectedString),
	characterCount => expectedCharacterCount
);	
assertionIsWrong := ((
		CNM_UnicodeUtilities.FindInUtf8String(
			ADR(upperStringToTest),
			ADR(upperExpectedString)
		) <> 1 
	) AND (
		expectedCharacterCount <> 0
	)
);

message := SEL(
	assertionIsWrong,
	'stringToCheck is $'%s$' start is $'%s$' assertion must be TRUE', 
	'stringToCheck is $'%s$' start is $'%s$' assertion must be FALSE'
);

IF (
		Tc2_Standard.LEN(stringToTest) = TO_UINT(Tc2_System.MAX_STRING_LENGTH)
) THEN
	stringToTestAsString := 'String with Tc2_System.MAX_STRING_LENGTH characters';
END_IF
IF (
		Tc2_Standard.LEN(expectedString) = TO_UINT(Tc2_System.MAX_STRING_LENGTH)
) THEN
	expectedStringAsString := 'String with Tc2_System.MAX_STRING_LENGTH characters';
END_IF

messageStringBuilder(
	sFormat := message,
	arg1 := THIS^.AnyToArg(stringToTestAsString),
	arg2 := THIS^.AnyToArg(expectedStringAsString)
);


THIS^.assertorContainer.assertor.assert.strings.unicode.startsWith(
	stringToCheck := stringToTest,
	start := expectedString,
	ignoreCases := TRUE,
	trim := FALSE,
	message			:= ''
);

THIS^.AssertEquals_BOOL(
	Expected 	:= assertionIsWrong,
	Actual 		:= THIS^.assertorContainer.wasAssertionWrong,
	Message 	:= messageStringBuilder.sOut
);

THIS^.AssertEquals_STRING(
	Expected 	:= stringToTestBeforeAssertion,
	Actual 		:= stringToTest,
	Message 	:= 'the assertion changed $'stringToTest$''
);

THIS^.AssertEquals_STRING(
	Expected 	:= expectedStringBeforeAssertion,
	Actual 		:= expectedString,
	Message 	:= 'the assertion changed $'expectedString$''
);

THIS^.assertorContainer.resetAssertor();

CNM_UnicodeUtilities.NormalizeUtf8String(
	utf8StringBuffer := ADR(stringToTest),
	bufferSize := Tc2_System.MAX_STRING_LENGTH + 1,
	normalizedStringBuffer := ADR(normalizedStringToTest),
	normalForm := CNM_UnicodeUtilities.NormalizationForm.NFD
);
CNM_UnicodeUtilities.NormalizeUtf8String(
	utf8StringBuffer := ADR(expectedString),
	bufferSize := Tc2_System.MAX_STRING_LENGTH + 1,
	normalizedStringBuffer := ADR(normalizedExpectedString),
	normalForm := CNM_UnicodeUtilities.NormalizationForm.NFD
);

normalizedUpperStringToTest := normalizedStringToTest;
normalizedUpperExpectedString := normalizedExpectedString;
CNM_UnicodeUtilities.UpperCaseUtf8(ADR(normalizedUpperStringToTest));
CNM_UnicodeUtilities.UpperCaseUtf8(ADR(normalizedUpperExpectedString));


CNM_UnicodeUtilities.GetUtf8StringLength(
	ADR(normalizedUpperExpectedString),
	characterCount => expectedCharacterCount
);
assertionIsWrong := ((
		CNM_UnicodeUtilities.FindInUtf8String(
			ADR(normalizedUpperStringToTest),
			ADR(normalizedUpperExpectedString),
		) <> 1
	) AND (
		expectedCharacterCount <> 0
	)
);

THIS^.assertorContainer.assertor.assert.strings.unicode.startsWith(
	stringToCheck := stringToTest,
	start := expectedString,
	ignoreCases := TRUE,
	trim		:= FALSE,
	normalizeStrings := TRUE,
	message			:= ''
);

THIS^.AssertEquals_BOOL(
	Expected 	:= assertionIsWrong,
	Actual 		:= THIS^.assertorContainer.wasAssertionWrong,
	Message 	:= messageStringBuilder.sOut
);

THIS^.AssertEquals_STRING(
	Expected 	:= stringToTestBeforeAssertion,
	Actual 		:= stringToTest,
	Message 	:= 'the assertion changed $'stringToTest$''
);

THIS^.AssertEquals_STRING(
	Expected 	:= expectedStringBeforeAssertion,
	Actual 		:= expectedString,
	Message 	:= 'the assertion changed $'expectedString$''
);
END_METHOD

(*
short summary
==================
This test method tests ``assert.string.unicode.startsWith``
method of CNM_AssertionInterfaces library with various inputs

.. <legal notes>

legal notes
=================
| SPDX-FileCopyrightText: © 2022 ekvip automation GmbH <info@ekvip.de>
| SPDX-License-Identifier: Apache-2.0
| For details check: Apache-2.0_

.. _Apache-2.0: https://www.apache.org/licenses/LICENSE-2.0

.. </legal notes>

*)


METHOD testStartsWithTrim : BOOL
VAR_INPUT
	(* for the test it's the parameter ``stringToCheck`` *)
	{attribute 'TcEncoding' := 'UTF-8'}
	stringToTest 	:Tc2_System.T_MaxString;
	(* for the test it's the parameter ``end`` *)
	{attribute 'TcEncoding' := 'UTF-8'}
	expectedString 	:Tc2_System.T_MaxString;
END_VAR
VAR 
	(* just the expectation if the assertion to test must be worng or true *)
	assertionIsWrong				:BOOL;
	(* contains the format string for the test message *)
	message							:Tc2_System.T_MaxString;
	(* contains trimed ´´stringToTest´´ *)
	trimedStringToTest				:Tc2_System.T_MaxString;
	(* contains trimed ´´expectedString´´ *)
	trimedExpectedString			:Tc2_System.T_MaxString;
	(* used for placeholder string if stringToTest can't be printed *)
	stringToTestAsString 			:Tc2_System.T_MaxString;
	(* used for placeholder string if expectedString can't be printed *)
	expectedStringAsString 			:Tc2_System.T_MaxString;
	(* contains stringToTest in normalized form *)
	normalizedStringToTest			:Tc2_System.T_MaxString;
	(* contains expectedString in normalized form *)
	normalizedExpectedString		:Tc2_System.T_MaxString;
	(* contains stringToTest in normalized form trimed *)
	normalizedTrimedStringToTest	:Tc2_System.T_MaxString;
	(* contains expectedString in normalized form trimed *)
	normalizedTrimedExpectedString	:Tc2_System.T_MaxString;
	(* holds characterCount of ``expectedString`` *)
	expectedCharacterCount			:UDINT;
	(* TwinCAT printf with the test message *)
	messageStringBuilder			:Tc2_Utilities.FB_FormatString;
	(* hold stringToCheck before assertion *)
	stringToTestBeforeAssertion		:Tc2_System.T_MaxString;
	(* hold expectedString before assertion *)
	expectedStringBeforeAssertion	:Tc2_System.T_MaxString;
END_VAR
THIS^.assertorContainer.resetAssertor();

stringToTestBeforeAssertion := stringToTest;
expectedStringBeforeAssertion := expectedString;
stringToTestAsString := stringToTest;
expectedStringAsString := expectedString;
trimedStringToTest := stringToTest;
trimedExpectedString := expectedString;

// trim the left of both strings
CNM_UnicodeUtilities.TrimLeftUtf8String(ADR(trimedStringToTest));
CNM_UnicodeUtilities.TrimLeftUtf8String(ADR(trimedExpectedString));

CNM_UnicodeUtilities.GetUtf8StringLength(
	ADR(trimedExpectedString),
	characterCount => expectedCharacterCount
);
assertionIsWrong := ((
		CNM_UnicodeUtilities.FindInUtf8String(
			ADR(trimedStringToTest),
			ADR(trimedExpectedString),
		) <> 1
	) AND (
		expectedCharacterCount <> 0
	)
);

message := SEL(
	assertionIsWrong,
	'stringToCheck is $'%s$' start is $'%s$' assertion must be TRUE', 
	'stringToCheck is $'%s$' start is $'%s$' assertion must be FALSE'
);

IF (
		Tc2_Standard.LEN(stringToTest) = TO_UINT(Tc2_System.MAX_STRING_LENGTH)
) THEN
	stringToTestAsString := 'String with Tc2_System.MAX_STRING_LENGTH characters';
END_IF
IF (
		Tc2_Standard.LEN(expectedString) = TO_UINT(Tc2_System.MAX_STRING_LENGTH)
) THEN
	expectedStringAsString := 'String with Tc2_System.MAX_STRING_LENGTH characters';
END_IF

messageStringBuilder(
	sFormat := message,
	arg1 := THIS^.AnyToArg(stringToTestAsString),
	arg2 := THIS^.AnyToArg(expectedStringAsString)
);


THIS^.assertorContainer.assertor.assert.strings.unicode.startsWith(
	stringToCheck := stringToTest,
	start := expectedString,
	ignoreCases := FALSE,
	trim := TRUE,
	normalizeStrings := FALSE,
	message			:= ''
);

THIS^.AssertEquals_BOOL(
	Expected 	:= assertionIsWrong,
	Actual 		:= THIS^.assertorContainer.wasAssertionWrong,
	Message 	:= messageStringBuilder.sOut
);

THIS^.AssertEquals_STRING(
	Expected 	:= stringToTestBeforeAssertion,
	Actual 		:= stringToTest,
	Message 	:= 'the assertion changed $'stringToTest$''
);

THIS^.AssertEquals_STRING(
	Expected 	:= expectedStringBeforeAssertion,
	Actual 		:= expectedString,
	Message 	:= 'the assertion changed $'expectedString$''
);

THIS^.assertorContainer.resetAssertor();

CNM_UnicodeUtilities.NormalizeUtf8String(
	utf8StringBuffer := ADR(stringToTest),
	bufferSize := Tc2_System.MAX_STRING_LENGTH + 1,
	normalizedStringBuffer := ADR(normalizedStringToTest),
	normalForm := CNM_UnicodeUtilities.NormalizationForm.NFD
);
CNM_UnicodeUtilities.NormalizeUtf8String(
	utf8StringBuffer := ADR(expectedString),
	bufferSize := Tc2_System.MAX_STRING_LENGTH + 1,
	normalizedStringBuffer := ADR(normalizedExpectedString),
	normalForm := CNM_UnicodeUtilities.NormalizationForm.NFD
);

normalizedTrimedStringToTest := normalizedStringToTest;
normalizedTrimedExpectedString := normalizedExpectedString;
CNM_UnicodeUtilities.TrimLeftUtf8String(ADR(normalizedTrimedStringToTest));
CNM_UnicodeUtilities.TrimLeftUtf8String(ADR(normalizedTrimedExpectedString));

CNM_UnicodeUtilities.GetUtf8StringLength(
	ADR(normalizedTrimedExpectedString),
	characterCount => expectedCharacterCount
);
assertionIsWrong := ((
		CNM_UnicodeUtilities.FindInUtf8String(
			ADR(normalizedTrimedStringToTest),
			ADR(normalizedTrimedExpectedString),
		) <> 1
	) AND (
		expectedCharacterCount <> 0
	)
);

THIS^.assertorContainer.assertor.assert.strings.unicode.startsWith(
	stringToCheck := stringToTest,
	start := expectedString,
	ignoreCases := FALSE,
	trim		:= TRUE,
	normalizeStrings := TRUE,
	message			:= ''
);

THIS^.AssertEquals_BOOL(
	Expected 	:= assertionIsWrong,
	Actual 		:= THIS^.assertorContainer.wasAssertionWrong,
	Message 	:= messageStringBuilder.sOut
);

THIS^.AssertEquals_STRING(
	Expected 	:= stringToTestBeforeAssertion,
	Actual 		:= stringToTest,
	Message 	:= 'the assertion changed $'stringToTest$''
);

THIS^.AssertEquals_STRING(
	Expected 	:= expectedStringBeforeAssertion,
	Actual 		:= expectedString,
	Message 	:= 'the assertion changed $'expectedString$''
);
END_METHOD

END_FUNCTION_BLOCK

// ---- AssertionTester/AssertionTests/StringAssertions/classes/Windows125xStringAssertionTests.TcPOU

(*
short summary
==================
This class tests all methods of Windows125x string assertions
with various combinations of inputs and checks expected 
outputs are satisfied or not

.. <legal notes>

legal notes
=================
| SPDX-FileCopyrightText: © 2022 ekvip automation GmbH <info@ekvip.de>
| SPDX-License-Identifier: Apache-2.0
| For details check: Apache-2.0_

.. _Apache-2.0: https://www.apache.org/licenses/LICENSE-2.0

.. </legal notes>

methods and properties
======================

*)


FUNCTION_BLOCK Windows125xStringAssertionTests EXTENDS AbstractAssertorTest
VAR
	
END_VAR
VAR CONSTANT
	(* prefix to unify the test names *)
	TEST_NAME_PREFIX :STRING := 'assert.string.windows125x.';
	
END_VAR

THIS^.runIsEmpty();
THIS^.runIsNotEmpty();
THIS^.runContains();
THIS^.runContainsNo();
THIS^.runEndsWith();
THIS^.runStartsWith();
THIS^.runIsEqualTo();
THIS^.runIsNotEqualTo();
THIS^.runLengthIsBetween();
THIS^.runLengthIsExact();
THIS^.runLengthIsMax();
THIS^.runLengthIsMin();

(*

short summary
==================
This test method is a helper function to create a unified test name

.. <legal notes>

legal notes
=================
| SPDX-FileCopyrightText: © 2022 ekvip automation GmbH <info@ekvip.de>
| SPDX-License-Identifier: Apache-2.0
| For details check: Apache-2.0_

.. _Apache-2.0: https://www.apache.org/licenses/LICENSE-2.0

.. </legal notes>

parameters
==========

*)

METHOD PROTECTED getTestNameFor :Tc2_System.T_MaxString
VAR_INPUT
	(* name of the method to test, to create a unified test name *)
	nameOfMethodToTest	:Tc2_System.T_MaxString;
END_VAR
getTestNameFor := Tc2_Standard.CONCAT(THIS^.TEST_NAME_PREFIX, nameOfMethodToTest);
END_METHOD

(*
short summary
==================
This test method tests ``assert.string.windows125x.contains``
method of CNM_AssertionInterfaces library with various inputs

.. <legal notes>

legal notes
=================
| SPDX-FileCopyrightText: © 2022 ekvip automation GmbH <info@ekvip.de>
| SPDX-License-Identifier: Apache-2.0
| For details check: Apache-2.0_

.. _Apache-2.0: https://www.apache.org/licenses/LICENSE-2.0

.. </legal notes>

*)


METHOD runContains : BOOL
VAR_INPUT
END_VAR
RETURN (NOT TcUnit.TEST_ORDERED(THIS^.getTestNameFor('contains')));

THIS^.testContains(
	stringToTest := '',
	expectedString := ''
);
THIS^.testContains(
	stringToTest := 'not empty',
	expectedString := ''
);
THIS^.testContains(
	stringToTest := '',
	expectedString := 'not empty'
);
THIS^.testContains(
	stringToTest := 'not empty',
	expectedString := 'not empty'
);
THIS^.testContains(
	stringToTest := '{|}~',
	expectedString := '3649213469328'
);
THIS^.testContains(
	stringToTest := '1one!',
	expectedString := '1'
);
THIS^.testContains(
	stringToTest := '1one!',
	expectedString := 'one'
);
THIS^.testContains(
	stringToTest := '1one!',
	expectedString := '!'
);
THIS^.testContains(
	stringToTest := '$40$n$t$$$"$'',
	expectedString := '$n$t'
);
THIS^.testContains(
	stringToTest := '$80$8C$A9$B9$C6$D4$F4$7E',
	expectedString := '$B9$C6$D4'
);
THIS^.testContains(
	stringToTest := '$80$8C$A9$B9$C6$D4$F4$7E',
	expectedString := '$80$B9$C6$D4'
);
THIS^.testContains(
	stringToTest := 'frontmiddleback',
	expectedString := 'back'
);
THIS^.testContains(
	stringToTest := 'frontmiddleback',
	expectedString := 'frontmiddlebackfront'
);
THIS^.testContains(
	stringToTest := 'backfrontmiddle',
	expectedString := 'backmiddle'
);
THIS^.testContains(
	stringToTest := 'J;%_iTxQSk?6GfWewt}yMKh1)VXqPA@P1YQ:{EAg:8VJ,/FM;j)xJ[[AvYp/}}SzEgtfYS,1K0.5VtA+VJrB(p#55h2z##mw#F)Y@P6Jz9G@6vb=x#E!cYk(Svr@S*KiPJr1VZ6AjrNback4G=vBJd.E:=,k3!wmuGDe#ZKMD#Vx%?M_0&L0#vT]J,+)ZvU{w%8X0=:XzthmT0VG0QrwpXXCWpFxu6[b!c.BunYYfLQi.,?ut?-{jrC1phTHL)y',
	expectedString := 'J;%_iTxQSk?6GfWewt}yMKh1)VXqPA@P1YQ:{EAg:8VJ,/FM;j)xJ[[AvYp/}}SzEgtfYS,1K0.5VtA+VJrB(p#55h2z##mw#F)Y@P6Jz9G@6vb=x#E!cYk(Svr@S*KiPJr1VZ6AjrNback4G=vBJd.E:=,k3!wmuGDe#ZKMD#Vx%?M_0&L0#vT]J,+)ZvU{w%8X0=:XzthmT0VG0QrwpXXCWpFxu6[b!c.BunYYfLQi.,?ut?-{jrC1phTHL)y'
);
THIS^.testContains(
	stringToTest := 'J;%_iTxQSk?6GfWewt}yMKh1)VXqPA@P1YQ:{EAg:8VJ,/FM;j)xJ[[AvYp/}}SzEgtfYS,1K0.5VtA+VJrB(p#55h2z##mw#F)Y@P6Jz9G@6vb=x#E!cYk(Svr@S*KiPJr1VZ6AjrNback4G=vBJd.E:=,k3!wmuGDe#ZKMD#Vx%?M_0&L0#vT]J,+)ZvU{w%8X0=:XzthmT0VG0QrwpXXCWpFxu6[b!c.BunYYfLQi.,?ut?-{jrC1phTHL)y',
	expectedString := 'J;%_iTxQSk?6GfWewt}yMKh1)VXqPA@P1YQ:{EAg:8VJ,/FM;j)xJ[[AvYp/}}SzEgtfYS,1K0.5VtA+VJrB(p#55h2z##mw#F)Y@P6Jz9G@6vb=x#E!cYk(Svr@S*KiPJr1VZ6AjrNback4G=vBJd.E:=,k3!wmuGDe#ZKMD#Vx%?M_0&L0#vT]J,+)ZvU{w%8X0=:XzthmT0VG0QrwpXXCWpFxu6[b!c.BunYYfLQi.,?ut?-{jrC1phTHL)x'
);

THIS^.testContainsIgnoreCase(
	stringToTest := 'UPPERCASE',
	expectedString := 'CASE'
);
THIS^.testContainsIgnoreCase(
	stringToTest := 'lowercase',
	expectedString := 'case'
);
THIS^.testContainsIgnoreCase(
	stringToTest := 'UPPERCASE',
	expectedString := 'case'
);
THIS^.testContainsIgnoreCase(
	stringToTest := 'lowercase',
	expectedString := 'CASE'
);
THIS^.testContainsIgnoreCase(
	stringToTest := 'lower',
	expectedString := 'UPPER'
);
THIS^.testContainsIgnoreCase(
	stringToTest := 'lowercase$80$B9$C6$D4',
	expectedString := 'CASE$80$B9$C6$D4'
);

TcUnit.TEST_FINISHED();
END_METHOD

(*
short summary
==================
This test method tests ``assert.string.windows125x.containsNo``
method of CNM_AssertionInterfaces library with various inputs

.. <legal notes>

legal notes
=================
| SPDX-FileCopyrightText: © 2022 ekvip automation GmbH <info@ekvip.de>
| SPDX-License-Identifier: Apache-2.0
| For details check: Apache-2.0_

.. _Apache-2.0: https://www.apache.org/licenses/LICENSE-2.0

.. </legal notes>

*)


METHOD runContainsNo : BOOL
RETURN (NOT TcUnit.TEST_ORDERED(THIS^.getTestNameFor('containsNo')));

THIS^.testContainsNo(
	stringToTest := '',
	expectedString := ''
);
THIS^.testContainsNo(
	stringToTest := 'not empty',
	expectedString := ''
);
THIS^.testContainsNo(
	stringToTest := '',
	expectedString := 'not empty'
);
THIS^.testContainsNo(
	stringToTest := 'not empty',
	expectedString := 'not empty'
);
THIS^.testContainsNo(
	stringToTest := '{|}~',
	expectedString := '3649213469328'
);
THIS^.testContainsNo(
	stringToTest := '1one!',
	expectedString := '1'
);
THIS^.testContainsNo(
	stringToTest := '1one!',
	expectedString := 'one'
);
THIS^.testContainsNo(
	stringToTest := '1one!',
	expectedString := '!'
);
THIS^.testContainsNo(
	stringToTest := '$40$n$t$$$"$'',
	expectedString := '$n$t'
);
THIS^.testContainsNo(
	stringToTest := '$80$8C$A9$B9$C6$D4$F4$7E',
	expectedString := '$B9$C6$D4'
);
THIS^.testContainsNo(
	stringToTest := '$80$8C$A9$B9$C6$D4$F4$7E',
	expectedString := '$80$B9$C6$D4'
);
THIS^.testContainsNo(
	stringToTest := 'frontmiddleback',
	expectedString := 'back'
);
THIS^.testContainsNo(
	stringToTest := 'frontmiddleback',
	expectedString := 'frontmiddlebackfront'
);
THIS^.testContainsNo(
	stringToTest := 'backfrontmiddle',
	expectedString := 'backmiddle'
);
THIS^.testContainsNo(
	stringToTest := 'J;%_iTxQSk?6GfWewt}yMKh1)VXqPA@P1YQ:{EAg:8VJ,/FM;j)xJ[[AvYp/}}SzEgtfYS,1K0.5VtA+VJrB(p#55h2z##mw#F)Y@P6Jz9G@6vb=x#E!cYk(Svr@S*KiPJr1VZ6AjrNback4G=vBJd.E:=,k3!wmuGDe#ZKMD#Vx%?M_0&L0#vT]J,+)ZvU{w%8X0=:XzthmT0VG0QrwpXXCWpFxu6[b!c.BunYYfLQi.,?ut?-{jrC1phTHL)y',
	expectedString := 'J;%_iTxQSk?6GfWewt}yMKh1)VXqPA@P1YQ:{EAg:8VJ,/FM;j)xJ[[AvYp/}}SzEgtfYS,1K0.5VtA+VJrB(p#55h2z##mw#F)Y@P6Jz9G@6vb=x#E!cYk(Svr@S*KiPJr1VZ6AjrNback4G=vBJd.E:=,k3!wmuGDe#ZKMD#Vx%?M_0&L0#vT]J,+)ZvU{w%8X0=:XzthmT0VG0QrwpXXCWpFxu6[b!c.BunYYfLQi.,?ut?-{jrC1phTHL)y'
);
THIS^.testContainsNo(
	stringToTest := 'J;%_iTxQSk?6GfWewt}yMKh1)VXqPA@P1YQ:{EAg:8VJ,/FM;j)xJ[[AvYp/}}SzEgtfYS,1K0.5VtA+VJrB(p#55h2z##mw#F)Y@P6Jz9G@6vb=x#E!cYk(Svr@S*KiPJr1VZ6AjrNback4G=vBJd.E:=,k3!wmuGDe#ZKMD#Vx%?M_0&L0#vT]J,+)ZvU{w%8X0=:XzthmT0VG0QrwpXXCWpFxu6[b!c.BunYYfLQi.,?ut?-{jrC1phTHL)y',
	expectedString := 'J;%_iTxQSk?6GfWewt}yMKh1)VXqPA@P1YQ:{EAg:8VJ,/FM;j)xJ[[AvYp/}}SzEgtfYS,1K0.5VtA+VJrB(p#55h2z##mw#F)Y@P6Jz9G@6vb=x#E!cYk(Svr@S*KiPJr1VZ6AjrNback4G=vBJd.E:=,k3!wmuGDe#ZKMD#Vx%?M_0&L0#vT]J,+)ZvU{w%8X0=:XzthmT0VG0QrwpXXCWpFxu6[b!c.BunYYfLQi.,?ut?-{jrC1phTHL)x'
);

THIS^.testContainsNoIgnoreCase(
	stringToTest := 'UPPERCASE',
	expectedString := 'CASE'
);
THIS^.testContainsNoIgnoreCase(
	stringToTest := 'lowercase',
	expectedString := 'case'
);
THIS^.testContainsNoIgnoreCase(
	stringToTest := 'UPPERCASE',
	expectedString := 'case'
);
THIS^.testContainsNoIgnoreCase(
	stringToTest := 'lowercase',
	expectedString := 'CASE'
);
THIS^.testContainsNoIgnoreCase(
	stringToTest := 'lower',
	expectedString := 'UPPER'
);
THIS^.testContainsNoIgnoreCase(
	stringToTest := 'lowercase$80$B9$C6$D4',
	expectedString := 'CASE$80$B9$C6$D4'
);

TcUnit.TEST_FINISHED();
END_METHOD

(*
short summary
==================
This test method tests ``assert.string.windows125x.endsWith``
method of CNM_AssertionInterfaces library with various inputs

.. <legal notes>

legal notes
=================
| SPDX-FileCopyrightText: © 2022 ekvip automation GmbH <info@ekvip.de>
| SPDX-License-Identifier: Apache-2.0
| For details check: Apache-2.0_

.. _Apache-2.0: https://www.apache.org/licenses/LICENSE-2.0

.. </legal notes>

*)


METHOD runEndsWith : BOOL
VAR_INPUT
END_VAR
RETURN (NOT TcUnit.TEST_ORDERED(THIS^.getTestNameFor('endsWith')));

THIS^.testEndsWith(
	stringToTest := '',
	expectedString := ''
);
THIS^.testEndsWith(
	stringToTest := 'not empty',
	expectedString := ''
);
THIS^.testEndsWith(
	stringToTest := '',
	expectedString := 'not empty'
);
THIS^.testEndsWith(
	stringToTest := 'not empty',
	expectedString := 'not empty'
);
THIS^.testEndsWith(
	stringToTest := '{|}~',
	expectedString := '3649213469328'
);
THIS^.testEndsWith(
	stringToTest := '1one!',
	expectedString := '1'
);
THIS^.testEndsWith(
	stringToTest := '1one!',
	expectedString := 'one'
);
THIS^.testEndsWith(
	stringToTest := '1one!',
	expectedString := '!'
);
THIS^.testEndsWith(
	stringToTest := '$40$n$t$$$"$'',
	expectedString := '$n$t'
);
THIS^.testEndsWith(
	stringToTest := '$40$$$"$'$n$t',
	expectedString := '$n$t'
);
THIS^.testEndsWith(
	stringToTest := '$80$8C$A9$B9$C6$D4$F4$7E',
	expectedString := '$B9$C6$D4'
);
THIS^.testEndsWith(
	stringToTest := '$80$8C$A9$B9$C6$D4$F4$7E',
	expectedString := '$80$B9$C6$D4'
);
THIS^.testEndsWith(
	stringToTest := 'frontmiddleback',
	expectedString := 'back'
);
THIS^.testEndsWith(
	stringToTest := 'frontmiddleback',
	expectedString := 'frontmiddlebackfront'
);
THIS^.testEndsWith(
	stringToTest := 'backfrontmiddle',
	expectedString := 'backmiddle'
);
THIS^.testEndsWith(
	stringToTest := 'J;%_iTxQSk?6GfWewt}yMKh1)VXqPA@P1YQ:{EAg:8VJ,/FM;j)xJ[[AvYp/}}SzEgtfYS,1K0.5VtA+VJrB(p#55h2z##mw#F)Y@P6Jz9G@6vb=x#E!cYk(Svr@S*KiPJr1VZ6AjrNback4G=vBJd.E:=,k3!wmuGDe#ZKMD#Vx%?M_0&L0#vT]J,+)ZvU{w%8X0=:XzthmT0VG0QrwpXXCWpFxu6[b!c.BunYYfLQi.,?ut?-{jrC1phTHL)y',
	expectedString := 'J;%_iTxQSk?6GfWewt}yMKh1)VXqPA@P1YQ:{EAg:8VJ,/FM;j)xJ[[AvYp/}}SzEgtfYS,1K0.5VtA+VJrB(p#55h2z##mw#F)Y@P6Jz9G@6vb=x#E!cYk(Svr@S*KiPJr1VZ6AjrNback4G=vBJd.E:=,k3!wmuGDe#ZKMD#Vx%?M_0&L0#vT]J,+)ZvU{w%8X0=:XzthmT0VG0QrwpXXCWpFxu6[b!c.BunYYfLQi.,?ut?-{jrC1phTHL)y'
);
THIS^.testEndsWith(
	stringToTest := 'J;%_iTxQSk?6GfWewt}yMKh1)VXqPA@P1YQ:{EAg:8VJ,/FM;j)xJ[[AvYp/}}SzEgtfYS,1K0.5VtA+VJrB(p#55h2z##mw#F)Y@P6Jz9G@6vb=x#E!cYk(Svr@S*KiPJr1VZ6AjrNback4G=vBJd.E:=,k3!wmuGDe#ZKMD#Vx%?M_0&L0#vT]J,+)ZvU{w%8X0=:XzthmT0VG0QrwpXXCWpFxu6[b!c.BunYYfLQi.,?ut?-{jrC1phTHL)y',
	expectedString := 'J;%_iTxQSk?6GfWewt}yMKh1)VXqPA@P1YQ:{EAg:8VJ,/FM;j)xJ[[AvYp/}}SzEgtfYS,1K0.5VtA+VJrB(p#55h2z##mw#F)Y@P6Jz9G@6vb=x#E!cYk(Svr@S*KiPJr1VZ6AjrNback4G=vBJd.E:=,k3!wmuGDe#ZKMD#Vx%?M_0&L0#vT]J,+)ZvU{w%8X0=:XzthmT0VG0QrwpXXCWpFxu6[b!c.BunYYfLQi.,?ut?-{jrC1phTHL)x'
);

THIS^.testEndsWithIgnoreCase(
	stringToTest := 'UPPERCASE',
	expectedString := 'CASE'
);
THIS^.testEndsWithIgnoreCase(
	stringToTest := 'lowercase',
	expectedString := 'case'
);
THIS^.testEndsWithIgnoreCase(
	stringToTest := 'UPPERCASE',
	expectedString := 'case'
);
THIS^.testEndsWithIgnoreCase(
	stringToTest := 'lowercase',
	expectedString := 'CASE'
);
THIS^.testEndsWithIgnoreCase(
	stringToTest := 'lower',
	expectedString := 'UPPER'
);
THIS^.testEndsWithIgnoreCase(
	stringToTest := 'lowercase$80$B9$C6$D4',
	expectedString := 'CASE$80$B9$C6$D4'
);

THIS^.testEndsWithTrim(
	stringToTest := 'frontmiddleback$t',
	expectedString := 'back',
	expectedAssertionResult := TRUE
);												
THIS^.testEndsWithTrim(
	stringToTest := 'frontmiddleback',
	expectedString := 'back$t',
	expectedAssertionResult := TRUE
);
THIS^.testEndsWithTrim(
	stringToTest := 'frontmiddleback$t',
	expectedString := 'back$t',
	expectedAssertionResult := TRUE
);
THIS^.testEndsWithTrim(
	stringToTest := 'frontmiddleback$20',
	expectedString := 'back',
	expectedAssertionResult := TRUE
);
THIS^.testEndsWithTrim(
	stringToTest := 'frontmiddleback',
	expectedString := 'back$20',
	expectedAssertionResult := TRUE
);
THIS^.testEndsWithTrim(
	stringToTest := 'frontmiddleback$t$n$r$p$l',
	expectedString := 'back',
	expectedAssertionResult := TRUE
);
THIS^.testEndsWithTrim(
	stringToTest := 'frontmiddleback$n$r$p$l',
	expectedString := 'back$25',
	expectedAssertionResult := FALSE
);												
THIS^.testEndsWithTrim(
	stringToTest := 'frontmiddleback$80$B9$C6$D4$20',
	expectedString := 'back$80$B9$C6$D4',
	expectedAssertionResult := TRUE
);
THIS^.testEndsWithTrim(
	stringToTest := 'frontmiddleback$80$B9$B9$C6$D4$20',
	expectedString := 'back$80$B9$C6$D4',
	expectedAssertionResult := FALSE
);

TcUnit.TEST_FINISHED();
END_METHOD

(*
short summary
==================
This test method tests ``assert.string.windows125x.IsEmpty``
method of CNM_AssertionInterfaces library with various inputs

.. <legal notes>

legal notes
=================
| SPDX-FileCopyrightText: © 2022 ekvip automation GmbH <info@ekvip.de>
| SPDX-License-Identifier: Apache-2.0
| For details check: Apache-2.0_

.. _Apache-2.0: https://www.apache.org/licenses/LICENSE-2.0

.. </legal notes>

*)


METHOD runIsEmpty : BOOL
VAR_INPUT
END_VAR
RETURN (NOT TcUnit.TEST_ORDERED(THIS^.getTestNameFor('IsEmpty')));

THIS^.testIsEmpty(
	stringToTest := ''
);
THIS^.testIsEmpty(
	stringToTest := 'not empty'
);
THIS^.testIsEmpty(
	stringToTest := '{|}~'
);
THIS^.testIsEmpty(
	stringToTest := '3649213469328'
);
THIS^.testIsEmpty(
	stringToTest := '1one!'
);
THIS^.testIsEmpty(
	stringToTest := '$40$n$t$$$"$''
);
THIS^.testIsEmpty(
	stringToTest := '$n$t'
);
THIS^.testIsEmpty(
	stringToTest := '$80$8C$A9$B9$C6$D4$F4$7E',
);
THIS^.testIsEmpty(
	stringToTest := 'frontmiddleback'
);
THIS^.testIsEmpty(
	stringToTest := 'backfrontmiddle'
);
THIS^.testIsEmpty(
	stringToTest := 'J;%_iTxQSk?6GfWewt}yMKh1)VXqPA@P1YQ:{EAg:8VJ,/FM;j)xJ[[AvYp/}}SzEgtfYS,1K0.5VtA+VJrB(p#55h2z##mw#F)Y@P6Jz9G@6vb=x#E!cYk(Svr@S*KiPJr1VZ6AjrNback4G=vBJd.E:=,k3!wmuGDe#ZKMD#Vx%?M_0&L0#vT]J,+)ZvU{w%8X0=:XzthmT0VG0QrwpXXCWpFxu6[b!c.BunYYfLQi.,?ut?-{jrC1phTHL)y'
);

TcUnit.TEST_FINISHED();
END_METHOD

(*
short summary
==================
This test method tests ``assert.string.windows125x.isEqualTo``
method of CNM_AssertionInterfaces library with various inputs

.. <legal notes>

legal notes
=================
| SPDX-FileCopyrightText: © 2022 ekvip automation GmbH <info@ekvip.de>
| SPDX-License-Identifier: Apache-2.0
| For details check: Apache-2.0_

.. _Apache-2.0: https://www.apache.org/licenses/LICENSE-2.0

.. </legal notes>

*)


METHOD runIsEqualTo : BOOL
VAR_INPUT
END_VAR
RETURN (NOT TcUnit.TEST_ORDERED(THIS^.getTestNameFor('isEqualTo')));

////////////////FAILING TESTS///////////////
(* 
-> SEE: ISSUE: #2 (https://ekv-app-git-p01.ekvip.de/CNMTC3/cnm4026/cnm4026-assertion-interface-lib/-/issues/2)
*)
////////////////////////////////////////////

THIS^.testisEqualTo(
	stringToTest := '',
	expectedString := ''
);
THIS^.testisEqualTo(
	stringToTest := 'not empty',
	expectedString := ''
);
THIS^.testisEqualTo(
	stringToTest := '',
	expectedString := 'not empty'
);
THIS^.testisEqualTo(
	stringToTest := 'not empty',
	expectedString := 'not'
);
THIS^.testisEqualTo(
	stringToTest := 'not empty',
	expectedString := 'not empty'
);
THIS^.testisEqualTo(
	stringToTest := '{|}~',
	expectedString := '3649213469328'
);
THIS^.testisEqualTo(
	stringToTest := '1one!',
	expectedString := '1one'
);
THIS^.testisEqualTo(
	stringToTest := '1one!',
	expectedString := '1one!'
);
THIS^.testisEqualTo(
	stringToTest := '$40$n$t$$$"$'',
	expectedString := '$n$t'
);
THIS^.testisEqualTo(
	stringToTest := '$40$n$t$$$"$'',
	expectedString := '$40$n$t$$$"$''
);
THIS^.testisEqualTo(
	stringToTest := '$80$8C$A9$B9$C6$D4$F4$7E',
	expectedString := '$B9$C6$D4'
);
THIS^.testisEqualTo(
	stringToTest := '$80$8C$A9$B9$C6$D4$F4$7E',
	expectedString := '$80$B9$C6$D4'
);
THIS^.testisEqualTo(
	stringToTest := 'frontmiddleback',
	expectedString := 'back'
);
THIS^.testisEqualTo(
	stringToTest := 'frontmiddleback',
	expectedString := 'frontmiddlebackfront'
);
THIS^.testisEqualTo(
	stringToTest := 'backfrontmiddle',
	expectedString := 'backmiddle'
);
THIS^.testisEqualTo(
	stringToTest := 'J;%_iTxQSk?6GfWewt}yMKh1)VXqPA@P1YQ:{EAg:8VJ,/FM;j)xJ[[AvYp/}}SzEgtfYS,1K0.5VtA+VJrB(p#55h2z##mw#F)Y@P6Jz9G@6vb=x#E!cYk(Svr@S*KiPJr1VZ6AjrNback4G=vBJd.E:=,k3!wmuGDe#ZKMD#Vx%?M_0&L0#vT]J,+)ZvU{w%8X0=:XzthmT0VG0QrwpXXCWpFxu6[b!c.BunYYfLQi.,?ut?-{jrC1phTHL)y',
	expectedString := 'J;%_iTxQSk?6GfWewt}yMKh1)VXqPA@P1YQ:{EAg:8VJ,/FM;j)xJ[[AvYp/}}SzEgtfYS,1K0.5VtA+VJrB(p#55h2z##mw#F)Y@P6Jz9G@6vb=x#E!cYk(Svr@S*KiPJr1VZ6AjrNback4G=vBJd.E:=,k3!wmuGDe#ZKMD#Vx%?M_0&L0#vT]J,+)ZvU{w%8X0=:XzthmT0VG0QrwpXXCWpFxu6[b!c.BunYYfLQi.,?ut?-{jrC1phTHL)y'
);
THIS^.testisEqualTo(
	stringToTest := 'J;%_iTxQSk?6GfWewt}yMKh1)VXqPA@P1YQ:{EAg:8VJ,/FM;j)xJ[[AvYp/}}SzEgtfYS,1K0.5VtA+VJrB(p#55h2z##mw#F)Y@P6Jz9G@6vb=x#E!cYk(Svr@S*KiPJr1VZ6AjrNback4G=vBJd.E:=,k3!wmuGDe#ZKMD#Vx%?M_0&L0#vT]J,+)ZvU{w%8X0=:XzthmT0VG0QrwpXXCWpFxu6[b!c.BunYYfLQi.,?ut?-{jrC1phTHL)y',
	expectedString := 'J;%_iTxQSk?6GfWewt}yMKh1)VXqPA@P1YQ:{EAg:8VJ,/FM;j)xJ[[AvYp/}}SzEgtfYS,1K0.5VtA+VJrB(p#55h2z##mw#F)Y@P6Jz9G@6vb=x#E!cYk(Svr@S*KiPJr1VZ6AjrNback4G=vBJd.E:=,k3!wmuGDe#ZKMD#Vx%?M_0&L0#vT]J,+)ZvU{w%8X0=:XzthmT0VG0QrwpXXCWpFxu6[b!c.BunYYfLQi.,?ut?-{jrC1phTHL)x'
);

